// TwinCAT 3 PLC project Plc
// libraries:
//   VisuElem3DPath, 3.5.6.0 (System)
//   VisuElemMeter, 3.5.6.0 (System)
//   VisuElems, 3.5.6.10 (System)
//   VisuElemsDateTime, 3.5.6.0 (System)
//   VisuElemsSpecialControls, 3.5.6.0 (System)
//   VisuElemsWinControls, 3.5.6.0 (System)
//   VisuElemTextEditor, 3.5.6.0 (System)
//   visuinputs, 3.5.6.0 (system)
//   VisuNativeControl, 3.5.6.0 (System)
//   Tc2_DMX, * (Beckhoff Automation GmbH)
//   Tc2_IoFunctions, * (Beckhoff Automation GmbH)
//   Tc2_Standard, * (Beckhoff Automation GmbH)
//   Tc2_SUPS, * (Beckhoff Automation GmbH)
//   Tc2_System, * (Beckhoff Automation GmbH)
//   Tc2_SystemCX, * (Beckhoff Automation GmbH)
//   Tc3_Interfaces, * (Beckhoff Automation GmbH)
//   Tc3_Module, * (Beckhoff Automation GmbH)
//   VisuDialogs, * (System)
//   Tc2_Utilities,3.3.11.0,Beckhoff Automation GmbH
// project tree:
//   Data types/ E_ModeRGB.TcDUT, E_StateKompressor.TcDUT, E_RolloMode.TcDUT, E_StateAnalog.TcDUT, E_WeekDay.TcDUT, ST_AnalogScaling.TcDUT, ST_DMXRGBWCtrl.TcDUT, ST_TimeSwitchTimes.TcDUT
//   Global Variables/ Globale_Variablen.TcGVL
//   / GlobalImagePool.TcGIPO (not stored), GlobalTextList.TcGTLO, PlcTaskMain.TcTTO, Visualization Manager.TcVMO (not stored), VISU_TASK.TcTTO
//   Logger/DUTs/ ST_LogFilter.TcDUT, ST_LogMessage.TcDUT, ST_LogMessageVisu.TcDUT
//   Logger/ FB_FileWriteLogString.TcPOU, FB_Logger.TcPOU, FB_LoggerSetMsg.TcPOU, G_Logger.TcGVL
//   Logger/VISUs/ V_LoggerFilterBlack.TcVIS, V_LoggerFilterLine.TcVIS, V_LoggerFilterList.TcVIS, V_LoggerFilterWhite.TcVIS, V_LoggerModul.TcVIS, V_LoggerMsgLine.TcVIS
//   POUs/Abluftsteuerung/ FB_Abluftsteuerung.TcPOU
//   POUs/Abluftsteuerung/SubSysteme/ FB_SubAbluftMaschine.TcPOU, FB_SubAbluftTaster.TcPOU
//   POUs/EG/ FB_EGHalle.TcPOU, FB_EGBuero.TcPOU
//   POUs/KG_Raueme/ FB_WCRaum.TcPOU
//   POUs/Kompressor/ FB_KompressorSteuerung.TcPOU
//   POUs/Monitoring/ FB_LiquidMonitoring.TcPOU
//   POUs/Monitoring/Submodule/ FB_LiquidSensor.TcPOU, FB_Transor.TcPOU
//   POUs/ PLC_PRG.TcPOU
//   POUs/Temperaturen/ PRG_Temperaturen.TcPOU
//   POUs/_Grundfunktionen/ FB_Heizregler.TcPOU, FB_Heizregler_FBHR.TcPOU, FB_Kuehlregler_Kompr.TcPOU, FB_Licht.TcPOU, FB_LichtBewegungsmelder.TcPOU, FB_Rollo.TcPOU, FB_RolloGruppe.TcPOU, FB_Taster.TcPOU, FB_TasterProg.TcPOU, FB_TemperatureInput.TcPOU, FB_AnalogOutput.TcPOU, FB_TimeSwitch.TcPOU, F_diColorOfTemperature.TcPOU, F_RolDownTime.TcPOU, F_Scaling.TcPOU, F_SunRise.TcPOU
//   POUs/_Grundfunktionen/System/ FB_BK1250Diag.TcPOU, FB_SystemCX.TcPOU
//   Visualizations/Frames/ V_Dialog_Mob.TcVIS, V_Main_Mob.TcVIS, V_Main_PC.TcVIS
//   Visualizations/Module/ V_ECReset.TcVIS, V_LiquidSensorCfg.TcVIS, V_LiquidSensorState.TcVIS, V_LiquidTransorState.TcVIS, V_NumInputReal.TcVIS, V_RadioButton.TcVIS, V_TCReset.TcVIS, V_WCRaum.TcVIS, V_WeekDay.TcVIS, V_dwBitToggle.TcVIS, V_Heizung.TcVIS, V_Licht.TcVIS, V_Rol.TcVIS, V_RolGrp.TcVIS
//   Visualizations/ VisuStart.TcVIS, V_Monitoring.TcVIS, V_Logger.TcVIS, V_KomprWRG.TcVIS, V_Einstellungen.TcVIS
// real-time tasks:
//   TASK Main: cycle T#5ms, priority 21, ADS port 350
//   TASK VISU_TASK: cycle T#100000us, priority 30, ADS port 351
// I/O:
//   DEVICE Device 3 (COM Port) (disabled)
//   DEVICE Device 2 (NOV-DP-RAM) (disabled)
//   DEVICE Device 5 (CX-BK) (disabled)
//     Box 5 (CX-BK)
//   DEVICE Device 8 (RT-Ethernet Protocol) (disabled), AmsNetId 0.0.0.0.9.1
//   DEVICE CX5120 (CX-BK)
//     CXBK (CX-BK)
//   DEVICE Device 1 (EtherCAT)
// variable links:
//   Plc Instance <-> CX5120 (CX-BK)/CXBK (CX-BK)
//     PlcTaskMain Inputs/.gfbTemp11_Puffer4000_Brauchw.IiDataIn <-> AI01 Temp (KL3204)/Channel 1/Data In
//     PlcTaskMain Inputs/.gfbTemp11_Puffer4000_Brauchw.IusiState <-> AI01 Temp (KL3204)/Channel 1/State
//     PlcTaskMain Inputs/.gfbTemp12_Puffer4000_oben.IiDataIn <-> AI01 Temp (KL3204)/Channel 2/Data In
//     PlcTaskMain Inputs/.gfbTemp12_Puffer4000_oben.IusiState <-> AI01 Temp (KL3204)/Channel 2/State
//     PlcTaskMain Inputs/.gfbTemp13_Puffer4000_mitte.IiDataIn <-> AI01 Temp (KL3204)/Channel 3/Data In
//     PlcTaskMain Inputs/.gfbTemp13_Puffer4000_mitte.IusiState <-> AI01 Temp (KL3204)/Channel 3/State
//     PlcTaskMain Inputs/.gfbTemp14_Puffer4000_unten.IiDataIn <-> AI01 Temp (KL3204)/Channel 4/Data In
//     PlcTaskMain Inputs/.gfbTemp14_Puffer4000_unten.IusiState <-> AI01 Temp (KL3204)/Channel 4/State
//     PlcTaskMain Inputs/.gfbTemp21_PufferWohnh_oben.IiDataIn <-> AI02 Temp (KL3204)/Channel 1/Data In
//     PlcTaskMain Inputs/.gfbTemp21_PufferWohnh_oben.IusiState <-> AI02 Temp (KL3204)/Channel 1/State
//     PlcTaskMain Inputs/.gfbTemp22_PufferWohnh_unten.IiDataIn <-> AI02 Temp (KL3204)/Channel 2/Data In
//     PlcTaskMain Inputs/.gfbTemp22_PufferWohnh_unten.IusiState <-> AI02 Temp (KL3204)/Channel 2/State
//     PlcTaskMain Inputs/.gfbTemp23_PufferWerkst_oben.IiDataIn <-> AI02 Temp (KL3204)/Channel 3/Data In
//     PlcTaskMain Inputs/.gfbTemp23_PufferWerkst_oben.IusiState <-> AI02 Temp (KL3204)/Channel 3/State
//     PlcTaskMain Inputs/.gfbTemp24_PufferWerkst_unten.IiDataIn <-> AI02 Temp (KL3204)/Channel 4/Data In
//     PlcTaskMain Inputs/.gfbTemp24_PufferWerkst_unten.IusiState <-> AI02 Temp (KL3204)/Channel 4/State
//     PlcTaskMain Inputs/.gfbTemp31_KomprWRG_Ruecklauf.IiDataIn <-> AI03 Temp (KL3204)/Channel 1/Data In
//     PlcTaskMain Inputs/.gfbTemp31_KomprWRG_Ruecklauf.IusiState <-> AI03 Temp (KL3204)/Channel 1/State
//     PlcTaskMain Inputs/.gfbTemp32_KomprWRG_Vorlauf.IiDataIn <-> AI03 Temp (KL3204)/Channel 2/Data In
//     PlcTaskMain Inputs/.gfbTemp32_KomprWRG_Vorlauf.IusiState <-> AI03 Temp (KL3204)/Channel 2/State
//     PlcTaskMain Inputs/.gfbTemp33_WCDamen_Raum.IiDataIn <-> AI03 Temp (KL3204)/Channel 3/Data In
//     PlcTaskMain Inputs/.gfbTemp33_WCDamen_Raum.IusiState <-> AI03 Temp (KL3204)/Channel 3/State
//     PlcTaskMain Inputs/.gfbTemp34_WCHerren_Raum.IiDataIn <-> AI03 Temp (KL3204)/Channel 4/Data In
//     PlcTaskMain Inputs/.gfbTemp34_WCHerren_Raum.IusiState <-> AI03 Temp (KL3204)/Channel 4/State
//     PlcTaskMain Inputs/.gfbTemp41_Schluckbrunnen.IiDataIn <-> AI04 Temp (KL3204)/Channel 1/Data In
//     PlcTaskMain Inputs/.gfbTemp41_Schluckbrunnen.IusiState <-> AI04 Temp (KL3204)/Channel 1/State
//     PlcTaskMain Inputs/.gfbTemp42_Res.IiDataIn <-> AI04 Temp (KL3204)/Channel 2/Data In
//     PlcTaskMain Inputs/.gfbTemp43_Res.IiDataIn <-> AI04 Temp (KL3204)/Channel 3/Data In
//     PlcTaskMain Inputs/.gfbTemp44_Res.IiDataIn <-> AI04 Temp (KL3204)/Channel 4/Data In
//     PlcTaskMain Inputs/.gfbTemp42_Res.IusiState <-> AI04 Temp (KL3204)/Channel 2/State
//     PlcTaskMain Inputs/.gfbTemp43_Res.IusiState <-> AI04 Temp (KL3204)/Channel 3/State
//     PlcTaskMain Inputs/.gfbTemp44_Res.IusiState <-> AI04 Temp (KL3204)/Channel 4/State
//     PlcTaskMain Inputs/PLC_PRG.fbAbluftsteuerung1.fbAblMasch01.IbMaschineEin <-> DI04 (KL1408)/Channel 1/Input
//     PlcTaskMain Inputs/PLC_PRG.fbAbluftsteuerung2.fbAblMasch01.IbMaschineEin <-> DI04 (KL1408)/Channel 2/Input
//     PlcTaskMain Inputs/PLC_PRG.fbAbluftsteuerung1.fbAblTaster1.IbStart <-> DI04 (KL1408)/Channel 3/Input
//     PlcTaskMain Inputs/PLC_PRG.fbAbluftsteuerung2.fbAblTaster1.IbStart <-> DI04 (KL1408)/Channel 4/Input
//     PlcTaskMain Inputs/PLC_PRG.fbEGBuero.fbLichtBueroAssist.IbInBewegunsm <-> DI02 (KL1408)/Channel 6/Input
//     PlcTaskMain Inputs/PLC_PRG.fbEGBuero.fbLichtBueroChef.IbInBewegunsm <-> DI02 (KL1408)/Channel 5/Input
//     PlcTaskMain Inputs/PLC_PRG.fbEGBuero.fbLichtPausenraum.IbInBewegunsm <-> DI02 (KL1408)/Channel 4/Input
//     PlcTaskMain Inputs/PLC_PRG.fbEGHalle.IbRolloWindmesser <-> DI03 (KL1408)/Channel 5/Input
//     PlcTaskMain Inputs/PLC_PRG.fbEGHalle.fbLichtHalleAltbau.IbInBewegunsm <-> DI02 (KL1408)/Channel 2/Input
//     PlcTaskMain Inputs/PLC_PRG.fbEGHalle.fbLichtHalleAnbau.IbInBewegunsm <-> DI02 (KL1408)/Channel 3/Input
//     PlcTaskMain Inputs/PLC_PRG.fbEGHalle.fbLichtHalleNeubau.IbInBewegunsm <-> DI02 (KL1408)/Channel 1/Input
//     PlcTaskMain Inputs/PLC_PRG.fbKompressorSteuerung.IbStart <-> DI01 (KL1408)/Channel 5/Input
//     PlcTaskMain Inputs/PLC_PRG.fbKompressorSteuerung.IbStoerung <-> DI01 (KL1408)/Channel 7/Input
//     PlcTaskMain Inputs/PLC_PRG.fbKompressorSteuerung.IbStop <-> DI01 (KL1408)/Channel 6/Input
//     PlcTaskMain Inputs/PLC_PRG.fbKompressorSteuerung.fbAnalogOutUmwaelzpumpeWRG.IiDataIn <-> AO01 (KL4004)/Channel 1/Data In
//     PlcTaskMain Inputs/PLC_PRG.fbKompressorSteuerung.fbAnalogOutUmwaelzpumpeWRG.IusiState <-> AO01 (KL4004)/Channel 1/State
//     PlcTaskMain Inputs/PLC_PRG.fbWCDamen.IbLichtBewegungsmelder <-> DI03 (KL1408)/Channel 2/Input
//     PlcTaskMain Inputs/PLC_PRG.fbWCDamen.IbTasterHeizenStart <-> DI03 (KL1408)/Channel 1/Input
//     PlcTaskMain Inputs/PLC_PRG.fbWCHerren.IbLichtBewegungsmelder <-> DI03 (KL1408)/Channel 4/Input
//     PlcTaskMain Inputs/PLC_PRG.fbWCHerren.IbTasterHeizenStart <-> DI03 (KL1408)/Channel 3/Input
//     PlcTaskMain Outputs/.gfbTemp11_Puffer4000_Brauchw.QiDataOut <-> AI01 Temp (KL3204)/Channel 1/Data Out
//     PlcTaskMain Outputs/.gfbTemp11_Puffer4000_Brauchw.QusiCtrl <-> AI01 Temp (KL3204)/Channel 1/Ctrl
//     PlcTaskMain Outputs/.gfbTemp12_Puffer4000_oben.QiDataOut <-> AI01 Temp (KL3204)/Channel 2/Data Out
//     PlcTaskMain Outputs/.gfbTemp12_Puffer4000_oben.QusiCtrl <-> AI01 Temp (KL3204)/Channel 2/Ctrl
//     PlcTaskMain Outputs/.gfbTemp13_Puffer4000_mitte.QiDataOut <-> AI01 Temp (KL3204)/Channel 3/Data Out
//     PlcTaskMain Outputs/.gfbTemp13_Puffer4000_mitte.QusiCtrl <-> AI01 Temp (KL3204)/Channel 3/Ctrl
//     PlcTaskMain Outputs/.gfbTemp14_Puffer4000_unten.QiDataOut <-> AI01 Temp (KL3204)/Channel 4/Data Out
//     PlcTaskMain Outputs/.gfbTemp14_Puffer4000_unten.QusiCtrl <-> AI01 Temp (KL3204)/Channel 4/Ctrl
//     PlcTaskMain Outputs/.gfbTemp21_PufferWohnh_oben.QiDataOut <-> AI02 Temp (KL3204)/Channel 1/Data Out
//     PlcTaskMain Outputs/.gfbTemp21_PufferWohnh_oben.QusiCtrl <-> AI02 Temp (KL3204)/Channel 1/Ctrl
//     PlcTaskMain Outputs/.gfbTemp22_PufferWohnh_unten.QiDataOut <-> AI02 Temp (KL3204)/Channel 2/Data Out
//     PlcTaskMain Outputs/.gfbTemp22_PufferWohnh_unten.QusiCtrl <-> AI02 Temp (KL3204)/Channel 2/Ctrl
//     PlcTaskMain Outputs/.gfbTemp23_PufferWerkst_oben.QiDataOut <-> AI02 Temp (KL3204)/Channel 3/Data Out
//     PlcTaskMain Outputs/.gfbTemp23_PufferWerkst_oben.QusiCtrl <-> AI02 Temp (KL3204)/Channel 3/Ctrl
//     PlcTaskMain Outputs/.gfbTemp24_PufferWerkst_unten.QiDataOut <-> AI02 Temp (KL3204)/Channel 4/Data Out
//     PlcTaskMain Outputs/.gfbTemp24_PufferWerkst_unten.QusiCtrl <-> AI02 Temp (KL3204)/Channel 4/Ctrl
//     PlcTaskMain Outputs/.gfbTemp31_KomprWRG_Ruecklauf.QiDataOut <-> AI03 Temp (KL3204)/Channel 1/Data Out
//     PlcTaskMain Outputs/.gfbTemp31_KomprWRG_Ruecklauf.QusiCtrl <-> AI03 Temp (KL3204)/Channel 1/Ctrl
//     PlcTaskMain Outputs/.gfbTemp32_KomprWRG_Vorlauf.QiDataOut <-> AI03 Temp (KL3204)/Channel 2/Data Out
//     PlcTaskMain Outputs/.gfbTemp32_KomprWRG_Vorlauf.QusiCtrl <-> AI03 Temp (KL3204)/Channel 2/Ctrl
//     PlcTaskMain Outputs/.gfbTemp33_WCDamen_Raum.QiDataOut <-> AI03 Temp (KL3204)/Channel 3/Data Out
//     PlcTaskMain Outputs/.gfbTemp33_WCDamen_Raum.QusiCtrl <-> AI03 Temp (KL3204)/Channel 3/Ctrl
//     PlcTaskMain Outputs/.gfbTemp34_WCHerren_Raum.QiDataOut <-> AI03 Temp (KL3204)/Channel 4/Data Out
//     PlcTaskMain Outputs/.gfbTemp34_WCHerren_Raum.QusiCtrl <-> AI03 Temp (KL3204)/Channel 4/Ctrl
//     PlcTaskMain Outputs/.gfbTemp41_Schluckbrunnen.QiDataOut <-> AI04 Temp (KL3204)/Channel 1/Data Out
//     PlcTaskMain Outputs/.gfbTemp41_Schluckbrunnen.QusiCtrl <-> AI04 Temp (KL3204)/Channel 1/Ctrl
//     PlcTaskMain Outputs/.gfbTemp42_Res.QiDataOut <-> AI04 Temp (KL3204)/Channel 2/Data Out
//     PlcTaskMain Outputs/.gfbTemp43_Res.QiDataOut <-> AI04 Temp (KL3204)/Channel 3/Data Out
//     PlcTaskMain Outputs/.gfbTemp44_Res.QiDataOut <-> AI04 Temp (KL3204)/Channel 4/Data Out
//     PlcTaskMain Outputs/.gfbTemp42_Res.QusiCtrl <-> AI04 Temp (KL3204)/Channel 2/Ctrl
//     PlcTaskMain Outputs/.gfbTemp43_Res.QusiCtrl <-> AI04 Temp (KL3204)/Channel 3/Ctrl
//     PlcTaskMain Outputs/.gfbTemp44_Res.QusiCtrl <-> AI04 Temp (KL3204)/Channel 4/Ctrl
//     PlcTaskMain Outputs/PLC_PRG.fbAbluftsteuerung1.QbAbluftVentilator <-> DO02 (KL2408)/Channel 5/Output
//     PlcTaskMain Outputs/PLC_PRG.fbAbluftsteuerung2.QbAbluftVentilator <-> DO02 (KL2408)/Channel 6/Output
//     PlcTaskMain Outputs/PLC_PRG.fbEGBuero.fbLichtBueroAssist.QbOutLicht <-> DO04 (KL2408)/Channel 7/Output
//     PlcTaskMain Outputs/PLC_PRG.fbEGBuero.fbLichtBueroChef.QbOutLicht <-> DO04 (KL2408)/Channel 6/Output
//     PlcTaskMain Outputs/PLC_PRG.fbEGHalle.QbRolloZentralAb <-> DO04 (KL2408)/Channel 2/Output
//     PlcTaskMain Outputs/PLC_PRG.fbEGHalle.QbRolloZentralAuf <-> DO04 (KL2408)/Channel 1/Output
//     PlcTaskMain Outputs/PLC_PRG.fbEGHalle.fbLichtHalleAltbau.QbOutLicht <-> DO04 (KL2408)/Channel 4/Output
//     PlcTaskMain Outputs/PLC_PRG.fbEGHalle.fbLichtHalleAnbau.QbOutLicht <-> DO04 (KL2408)/Channel 5/Output
//     PlcTaskMain Outputs/PLC_PRG.fbEGHalle.fbLichtHalleNeubau.QbOutLicht <-> DO04 (KL2408)/Channel 3/Output
//     PlcTaskMain Outputs/PLC_PRG.fbKompressorSteuerung.QbKompressor <-> DO01 (KL2408)/Channel 6/Output
//     PlcTaskMain Outputs/PLC_PRG.fbKompressorSteuerung.QbLMStatus <-> DO01 (KL2408)/Channel 5/Output
//     PlcTaskMain Outputs/PLC_PRG.fbKompressorSteuerung.QbLufttrockner <-> DO01 (KL2408)/Channel 8/Output
//     PlcTaskMain Outputs/PLC_PRG.fbKompressorSteuerung.QbNotKompressor <-> DO01 (KL2408)/Channel 7/Output
//     PlcTaskMain Outputs/PLC_PRG.fbKompressorSteuerung.QbUmwaelzpumpeWRG <-> DO02 (KL2408)/Channel 1/Output
//     PlcTaskMain Outputs/PLC_PRG.fbKompressorSteuerung.QbUmwaelzpumpeWohnhaus <-> DO02 (KL2408)/Channel 3/Output
//     PlcTaskMain Outputs/PLC_PRG.fbKompressorSteuerung.QbVentilSchnellauflWRG <-> DO02 (KL2408)/Channel 2/Output
//     PlcTaskMain Outputs/PLC_PRG.fbKompressorSteuerung.QbVentilUmschWerkstatt <-> DO02 (KL2408)/Channel 4/Output
//     PlcTaskMain Outputs/PLC_PRG.fbKompressorSteuerung.fbAnalogOutUmwaelzpumpeWRG.QiDataOut <-> AO01 (KL4004)/Channel 1/Data Out
//     PlcTaskMain Outputs/PLC_PRG.fbKompressorSteuerung.fbAnalogOutUmwaelzpumpeWRG.QusiCtrl <-> AO01 (KL4004)/Channel 1/Ctrl
//     PlcTaskMain Outputs/PLC_PRG.fbWCDamen.QbAbluftventilator <-> DO03 (KL2408)/Channel 3/Output
//     PlcTaskMain Outputs/PLC_PRG.fbWCDamen.QbLMHeizungAktiv <-> DO03 (KL2408)/Channel 1/Output
//     PlcTaskMain Outputs/PLC_PRG.fbWCDamen.QbStellventilHeizkoerper <-> DO03 (KL2408)/Channel 2/Output
//     PlcTaskMain Outputs/PLC_PRG.fbWCHerren.QbAbluftventilator <-> DO03 (KL2408)/Channel 6/Output
//     PlcTaskMain Outputs/PLC_PRG.fbWCHerren.QbLMHeizungAktiv <-> DO03 (KL2408)/Channel 4/Output
//     PlcTaskMain Outputs/PLC_PRG.fbWCHerren.QbStellventilHeizkoerper <-> DO03 (KL2408)/Channel 5/Output
//   Plc Instance <-> Device 1 (EtherCAT)
//     PlcTaskMain Inputs/.gfbSystemCX.IuiDevState_ECMAster <-> Inputs/DevState
//   Plc Instance <-> Device 1 (EtherCAT)/Box 1 (BK1150)
//     PlcTaskMain Inputs/PLC_PRG.fbLiquidMonitoring.IbContactorResponse1 <-> DI12 (KL1408)/Channel 2/Input
//     PlcTaskMain Inputs/PLC_PRG.fbLiquidMonitoring.IbContactorResponse2 <-> DI12 (KL1408)/Channel 3/Input
//     PlcTaskMain Inputs/PLC_PRG.fbLiquidMonitoring.IbStartQuit <-> DI12 (KL1408)/Channel 1/Input
//     PlcTaskMain Inputs/PLC_PRG.fbLiquidMonitoring.fbLiquidSensor[10].IbLiquidSensor <-> DI13 (KL1408)/Channel 5/Input
//     PlcTaskMain Inputs/PLC_PRG.fbLiquidMonitoring.fbLiquidSensor[11].IbLiquidSensor <-> DI13 (KL1408)/Channel 6/Input
//     PlcTaskMain Inputs/PLC_PRG.fbLiquidMonitoring.fbLiquidSensor[12].IbLiquidSensor <-> DI13 (KL1408)/Channel 7/Input
//     PlcTaskMain Inputs/PLC_PRG.fbLiquidMonitoring.fbLiquidSensor[1].IbLiquidSensor <-> DI12 (KL1408)/Channel 4/Input
//     PlcTaskMain Inputs/PLC_PRG.fbLiquidMonitoring.fbLiquidSensor[2].IbLiquidSensor <-> DI12 (KL1408)/Channel 5/Input
//     PlcTaskMain Inputs/PLC_PRG.fbLiquidMonitoring.fbLiquidSensor[3].IbLiquidSensor <-> DI12 (KL1408)/Channel 6/Input
//     PlcTaskMain Inputs/PLC_PRG.fbLiquidMonitoring.fbLiquidSensor[4].IbLiquidSensor <-> DI12 (KL1408)/Channel 7/Input
//     PlcTaskMain Inputs/PLC_PRG.fbLiquidMonitoring.fbLiquidSensor[5].IbLiquidSensor <-> DI12 (KL1408)/Channel 8/Input
//     PlcTaskMain Inputs/PLC_PRG.fbLiquidMonitoring.fbLiquidSensor[6].IbLiquidSensor <-> DI13 (KL1408)/Channel 1/Input
//     PlcTaskMain Inputs/PLC_PRG.fbLiquidMonitoring.fbLiquidSensor[7].IbLiquidSensor <-> DI13 (KL1408)/Channel 2/Input
//     PlcTaskMain Inputs/PLC_PRG.fbLiquidMonitoring.fbLiquidSensor[8].IbLiquidSensor <-> DI13 (KL1408)/Channel 3/Input
//     PlcTaskMain Inputs/PLC_PRG.fbLiquidMonitoring.fbLiquidSensor[9].IbLiquidSensor <-> DI13 (KL1408)/Channel 4/Input
//     PlcTaskMain Outputs/PLC_PRG.fbLiquidMonitoring.QbLMStartQuit <-> DO12 (KL2408)/Channel 7/Output
//     PlcTaskMain Outputs/PLC_PRG.fbLiquidMonitoring.QbLMStatusOK <-> DO12 (KL2408)/Channel 6/Output
//     PlcTaskMain Outputs/PLC_PRG.fbLiquidMonitoring.QbStartTransor <-> DO12 (KL2408)/Channel 1/Output
//     PlcTaskMain Outputs/PLC_PRG.fbLiquidMonitoring.fbLiquidSensor[10].QbLMStatus <-> DO14 (KL2408)/Channel 2/Output
//     PlcTaskMain Outputs/PLC_PRG.fbLiquidMonitoring.fbLiquidSensor[11].QbLMStatus <-> DO14 (KL2408)/Channel 3/Output
//     PlcTaskMain Outputs/PLC_PRG.fbLiquidMonitoring.fbLiquidSensor[12].QbLMStatus <-> DO14 (KL2408)/Channel 4/Output
//     PlcTaskMain Outputs/PLC_PRG.fbLiquidMonitoring.fbLiquidSensor[1].QbLMStatus <-> DO13 (KL2408)/Channel 1/Output
//     PlcTaskMain Outputs/PLC_PRG.fbLiquidMonitoring.fbLiquidSensor[2].QbLMStatus <-> DO13 (KL2408)/Channel 2/Output
//     PlcTaskMain Outputs/PLC_PRG.fbLiquidMonitoring.fbLiquidSensor[3].QbLMStatus <-> DO13 (KL2408)/Channel 3/Output
//     PlcTaskMain Outputs/PLC_PRG.fbLiquidMonitoring.fbLiquidSensor[4].QbLMStatus <-> DO13 (KL2408)/Channel 4/Output
//     PlcTaskMain Outputs/PLC_PRG.fbLiquidMonitoring.fbLiquidSensor[5].QbLMStatus <-> DO13 (KL2408)/Channel 5/Output
//     PlcTaskMain Outputs/PLC_PRG.fbLiquidMonitoring.fbLiquidSensor[6].QbLMStatus <-> DO13 (KL2408)/Channel 6/Output
//     PlcTaskMain Outputs/PLC_PRG.fbLiquidMonitoring.fbLiquidSensor[7].QbLMStatus <-> DO13 (KL2408)/Channel 7/Output
//     PlcTaskMain Outputs/PLC_PRG.fbLiquidMonitoring.fbLiquidSensor[8].QbLMStatus <-> DO13 (KL2408)/Channel 8/Output
//     PlcTaskMain Outputs/PLC_PRG.fbLiquidMonitoring.fbLiquidSensor[9].QbLMStatus <-> DO14 (KL2408)/Channel 1/Output
//     PlcTaskMain Outputs/PLC_PRG.fbLiquidMonitoring.fbTransor[{1..4}].QbTransor <-> DO12 (KL2408)/Channel {2..5}/Output  (4 links)

CONFIGURATION Plc
    RESOURCE PLC ON TwinCAT3
        TASK PlcTaskMain(INTERVAL := T#5ms, PRIORITY := 21);
        TASK VISU_TASK(INTERVAL := T#100000us, PRIORITY := 30);
        PROGRAM PLC_PRG WITH PlcTaskMain : PLC_PRG;
        PROGRAM VisuElems_Visu_Prg WITH VISU_TASK : VisuElems.Visu_Prg;
    END_RESOURCE
END_CONFIGURATION

// ---- Data types/E_ModeRGB.TcDUT
TYPE E_ModeRGB :
(
	eModeRGB_Off,
	eModeRGB_MANUAL,
	eModeRGB_AUTO,
	eModeRGB_AUTOREVERS
);
END_TYPE

// ---- Data types/E_StateKompressor.TcDUT
TYPE E_StateKompressor :
(
	eStateKompr_AUS,
	eStateKompr_START,
	eStateKompr_AKTIV,
	eStateKompr_STOP,
	eStateKompr_STOERUNG
);
END_TYPE

// ---- Data types/E_RolloMode.TcDUT
TYPE E_RolloMode : (
	eRollo_Stop,
	eRollo_Manuell,
	eRollo_Auto,
	eRollo_Schatten);
END_TYPE

// ---- Data types/E_StateAnalog.TcDUT
TYPE E_StateAnalog : (
	eAnalog_Init,
	eAnalog_Start,
	eAnalog_LimitLow,
	eAnalog_LimitHigh,
	eAnalog_End
	);
END_TYPE

// ---- Data types/E_WeekDay.TcDUT
TYPE E_WeekDay :(
	Sonntag,
	Montag,
	Dienstag,
	Mittwoch,
	Donnerstag,
	Freitag,
	Samstag,

// folgende Eintraege sind nur zur Moduloberechnung
	Sonntag2,
	Montag2,
	Dienstag2,
	Mittwoch2,
	Donnerstag2,
	Freitag2,
	Samstag2
	);
END_TYPE

// ---- Data types/ST_AnalogScaling.TcDUT
TYPE ST_AnalogScaling :
STRUCT
	diXRef 	: DINT := 0;
	diYRef	: DINT := 2100;
	diFact	: DINT := 5000;

END_STRUCT
END_TYPE

// ---- Data types/ST_DMXRGBWCtrl.TcDUT
TYPE ST_DMXRGBWCtrl :
STRUCT
	bTickManual		: BOOL; (* Zyklus-Ticks fuer manuelle Verstellung *)
	bTickAuto			: BOOL; (* Zyklus-Ticks fuer automatische Programme *)
	rBrightness		: REAL := 1.0; (* zentraler Helligkeits-Override *)
	rRGBCtrl			: REAL; (* Steuerwert fuer den Farbton *)
	byRed					: BYTE; (* Steuerwert fuer den Farbton rot *)
	byGreen				: BYTE; (* Steuerwert fuer den Farbton grün *)
	byBlue				: BYTE; (* Steuerwert fuer den Farbton blau *)
	byWhite				: BYTE; (* Steuerwert fuer den Farbton weiss *)
	
END_STRUCT
END_TYPE

// ---- Data types/ST_TimeSwitchTimes.TcDUT
TYPE ST_TimeSwitchTimes :
STRUCT
	todHeizEin		: ARRAY[0..iTIMESWITCH_NUMOFTIMES] OF TIME_OF_DAY;
	todHeizAus		: ARRAY[0..iTIMESWITCH_NUMOFTIMES] OF TIME_OF_DAY;
	eDayOfWeekStart : ARRAY[0..iTIMESWITCH_NUMOFTIMES] OF E_WeekDay := [iTIMESWITCH_NUMOFTIMES(Montag)];
	eDayOfWeekEnd : ARRAY[0..iTIMESWITCH_NUMOFTIMES] OF E_WeekDay := [iTIMESWITCH_NUMOFTIMES(Sonntag)];

END_STRUCT
END_TYPE

// ---- Logger/DUTs/ST_LogFilter.TcDUT
TYPE ST_LogFilter :
(*
  ***************************************************************************
  ***************************************************************************
  Module owner:                 ST_EW_SW_SY, woerz 
  Keyword:                      keyword, <Feature-ID> 
  
  Description (summary): PLC Message logger filter

  ***************************************************************************
*)
STRUCT
  bEnabled : BOOL;
  szText : STRING(40);
END_STRUCT
END_TYPE

// ---- Logger/DUTs/ST_LogMessage.TcDUT
TYPE ST_LogMessage :
STRUCT
  iTyp : INT; // 0=hint 1=warning 2=error
  dtDateTime : DATE_AND_TIME;
  szPath : STRING(60);
  szMessage : STRING(80);
END_STRUCT
END_TYPE

// ---- Logger/DUTs/ST_LogMessageVisu.TcDUT
TYPE ST_LogMessageVisu :
STRUCT
	iLogId : INT;
	iTyp : INT;
	szLogMsg : STRING(160);
END_STRUCT
END_TYPE

// ---- Global Variables/Globale_Variablen.TcGVL
{attribute 'Tc2GvlVarNames'}
VAR_GLOBAL CONSTANT
	gciHeizGr			: INT := 9;
	gciHeizTimer 	: INT := 1;
	giPWMMax			: INT := 150;
	gdwPWMfast_75 : DWORD := 2000;
	gdwPWMfast_88 : DWORD := 8000;

	giNumOfAICh		: INT := 6;
	giNumOfAIGrp	: INT := 7;

	iTIMESWITCH_NUMOFTIMES : INT := 5;

END_VAR

VAR_GLOBAL
	gbTakt100ms		: BOOL;
  gdwBlink      : DWORD;

	gfbSystemCX		: FB_SystemCX := (INCFGDiagBK1250:= TRUE);

	grSunRiseFact : REAL;

	gbLichtZentralAus 	: BOOL := FALSE;
	gbLichtZentralEin 	: BOOL := FALSE;

	gbTimeRolloAb				: BOOL;
	gbTimeRolloAuf			: BOOL;

	gbTimeNacht					: BOOL;
	gbTimeTag						: BOOL;
	gbTag								: BOOL;
	gbNacht							: BOOL := TRUE;

	gbPWMTakt						: BOOL;
	giPWMTimer					: INT;
	gbHeizGruppe 				: ARRAY[0..gciHeizGr] OF BOOL;

	(* Temperatureingänge *)
	gfbTemp11_Puffer4000_Brauchw	: FB_TemperatureInput := ( (*  *)
		INrCalibFactor := 1.0,
		INrCalibOffset := 0.0);
	gfbTemp12_Puffer4000_oben			: FB_TemperatureInput := ( (*  *)
		INrCalibFactor := 1.0,
		INrCalibOffset := 0.0);
	gfbTemp13_Puffer4000_mitte		: FB_TemperatureInput := ( (*  *)
		INrCalibFactor := 1.0,
		INrCalibOffset := 0.0);
	gfbTemp14_Puffer4000_unten		: FB_TemperatureInput := ( (*  *)
		INrCalibFactor := 1.0,
		INrCalibOffset := 0.0);
	gfbTemp21_PufferWohnh_oben	: FB_TemperatureInput := ( (*  *)
		INrCalibFactor := 1.0,
		INrCalibOffset := 0.0);
	gfbTemp22_PufferWohnh_unten		: FB_TemperatureInput := ( (*  *)
		INrCalibFactor := 1.0,
		INrCalibOffset := 0.0);
	gfbTemp23_PufferWerkst_oben		: FB_TemperatureInput := ( (*  *)
		INrCalibFactor := 1.0,
		INrCalibOffset := 0.0);
	gfbTemp24_PufferWerkst_unten	: FB_TemperatureInput := ( (*  *)
		INrCalibFactor := 1.0,
		INrCalibOffset := 0.0);
	gfbTemp31_KomprWRG_Ruecklauf	: FB_TemperatureInput := ( (* Wassertemperatur WRG zum Puffer (heiss) *)
		INrCalibFactor := 1.0,
		INrCalibOffset := 0.0);
	gfbTemp32_KomprWRG_Vorlauf		: FB_TemperatureInput := ( (*  *)
		INrCalibFactor := 1.0,
		INrCalibOffset := 0.0);
	gfbTemp33_WCDamen_Raum				: FB_TemperatureInput := ( (*  *)
		INrCalibFactor := 1.0,
		INrCalibOffset := 0.0);
	gfbTemp34_WCHerren_Raum				: FB_TemperatureInput := ( (*  *)
		INrCalibFactor := 1.0,
		INrCalibOffset := 0.0);
	gfbTemp41_Schluckbrunnen			: FB_TemperatureInput := ( (*  *)
		INrCalibFactor := 1.0,
		INrCalibOffset := 0.0);
	gfbTemp42_Res									: FB_TemperatureInput := ( (*  *)
		INrCalibFactor := 1.0,
		INrCalibOffset := 0.0);
	gfbTemp43_Res									: FB_TemperatureInput := ( (*  *)
		INrCalibFactor := 1.0,
		INrCalibOffset := 0.0);
	gfbTemp44_Res									: FB_TemperatureInput := ( (*  *)
		INrCalibFactor := 1.0,
		INrCalibOffset := 0.0);

END_VAR

VAR_GLOBAL PERSISTENT
	VnvdiLichtTofKurz	: DINT := 5; (* Minuten *)
	VnvdiLichtTofLang	: DINT := 60; (* Minuten *)
	VnvstSwitchTimesLichtBWMtofLang : ST_TimeSwitchTimes; // Bewegungsmelder-Licht: Schaltzeiten fuer lange Ausschaltverzoegerung 

END_VAR

// ---- Logger/G_Logger.TcGVL
(*
  ***************************************************************************
  ***************************************************************************
  Module owner:                 ST_EW_SW_SY, woerz 
  Keyword:                      keyword, <Feature-ID> 
  
  Description (summary): PLC Message logger

  ***************************************************************************
*)
VAR_GLOBAL CONSTANT
  iMAXNUMOFMSGPERSISTENT : INT := 500; // maximum num of messages in persistent array
  iMINNUMOFMSGWRITETOFILE : INT := 100; // writing to file will start, if this num of messages are present
  iMINTIMEAFTERFILEWRITING : TIME := T#10M; // minimum waiting time, after writing to file
  iMAXNUMOFLOGFILES : INT := 3; // maximum num of log files
  diMAXNUMOFLOGITEMSPERFILE : DINT := 5000; // maximum num of log items per file
  
   // file path/name on target system (IPC)
  szLOGFILEPATH_TARGETSYSTEM : T_MaxString := 'C:\PlcLogger\'; ; 
  szLOGFILEPATH_NETWORK : T_MaxString := 'S:\Dokumente\PlcLogger\';
  
END_VAR
VAR_GLOBAL
  gfbLogger : FB_Logger;

END_VAR

// ---- POUs/PLC_PRG.TcPOU
PROGRAM PLC_PRG
VAR
	bInit							: BOOL := TRUE;

	tonCount : TON := (PT:= t#200ms);

	bSetClock  				: BOOL;
	bCopyToClockSet 	: BOOL := TRUE;
	bTimeCalc  				: BOOL;
	dtClockSet 				: DATE_AND_TIME := DT#2008-01-01-00:00;
	dwSysTimeSet			: DWORD;

	rtrigRolloAb	: R_TRIG;
	rtrigRolloAuf : R_TRIG;
	bVisuRolloAb 	: BOOL;
	bVisuRolloAuf : BOOL;

	tonTakt100ms	: TON := (PT:= t#100ms);
	tonTaktPWM	: TON := (PT:= t#5s);
	bTakt200ms	: BOOL;

	todRolloAb_i		: TIME_OF_DAY;

	dwdNacht_i			: DWORD;
	todNacht_i			: TIME_OF_DAY;
	todTag_i				: TIME_OF_DAY;

	bIn										: BOOL;
	fbTasterZentral1 			: FB_Taster;
	IbZentral1  	 AT %I* : BOOL;
	bInVisuZentral1				: BOOL;

	bVisuLichtZentralAus 	: BOOL;
	bVisuLichtZentralEin 	: BOOL;

	bLichtZentralAus 	: BOOL;
	bLichtZentralEin 	: BOOL;

(*
	fbTasterZentral2 		: FB_Taster;
	IbZentral2  AT %I*3.1	: BOOL;
	bInVisuZentral2			: BOOL;*)

	iHGr	: INT;
	iHTi	: INT;
	
	(* Funktionsbausteine ************************************)

	(* Kompressorsteuerung ***********************************)
	fbKompressorSteuerung		: FB_KompressorSteuerung;

	(* Abluft bzw. Absaugung *********************************)
	fbAbluftsteuerung1			: FB_Abluftsteuerung;
	fbAbluftsteuerung2			: FB_Abluftsteuerung;
	
  // Monitoring
  fbLiquidMonitoring : FB_LiquidMonitoring;

	(* EG-Raeume *)
  fbEGHalle : FB_EGHalle;
  fbEGBuero : FB_EGBuero;
  
	(* KG-Raeume *)
	fbWCDamen								: FB_WCRaum();
	fbWCHerren							: FB_WCRaum();
	
	
  fbLog : FB_LoggerSetMsg;
END_VAR

VAR PERSISTENT
	bSummerTime		: BOOL;

	todRolloAuf		: TIME_OF_DAY := TOD#7:30;
	todRolloAb		: TIME_OF_DAY := TOD#18:55;
	dwRolloAbMinFact_neg	: DWORD := 115;
	dwRolloAbMinFact_pos	: DWORD := 135;


	todHeizEin		: ARRAY[0..gciHeizGr,0..gciHeizTimer] OF TIME_OF_DAY :=[ TOD#0:00];
	todHeizAus		: ARRAY[0..gciHeizGr,0..gciHeizTimer] OF TIME_OF_DAY :=[ TOD#0:00];

END_VAR

IF bInit THEN
	A_Init();
END_IF
gfbSystemCX();


(* Systemuhr ***************************)
IF gfbSystemCX.OUTbNewDay
OR bTimeCalc
THEN
	(* Datum hat sich geaendert (neuer Tag) *)
	A_TimeCalculation();
	bTimeCalc := FALSE;
END_IF

(* Rollo-Timer *)
IF (todRolloAb <> TOD#00:00) THEN
	rtrigRolloAb(CLK:= (gfbSystemCX.OUTtodClockBase = todRolloAb_i));
  IF rtrigRolloAb.Q OR bVisuRolloAb THEN
    IF NOT gbTimeRolloAb THEN
      fbLog.M_AddMsgHint('Rollo AB zentral');
    END_IF
	  gbTimeRolloAb := TRUE;
	END_IF
ELSE
	gbTimeRolloAb := FALSE;
END_IF
IF (todRolloAuf <> TOD#00:00) THEN
	rtrigRolloAuf(CLK:= (gfbSystemCX.OUTtodClock = todRolloAuf));
  IF rtrigRolloAuf.Q OR bVisuRolloAuf THEN
    IF NOT gbTimeRolloAuf THEN
      fbLog.M_AddMsgHint('Rollo AUF zentral');
    END_IF
	  gbTimeRolloAuf := TRUE;
	END_IF
ELSE
	gbTimeRolloAuf := FALSE;
END_IF


(* Tag/Nacht-Timer *)
gbTimeNacht := FALSE;
gbTimeTag := FALSE;
IF (gfbSystemCX.OUTtodClockBase = todTag_i) THEN
	gbTimeTag := TRUE;
	gbTag := TRUE;
	gbNacht := FALSE;
ELSIF (gfbSystemCX.OUTtodClockBase = todNacht_i) THEN
	gbTimeNacht := TRUE;
	gbTag := FALSE;
	gbNacht := TRUE;
END_IF



(* Heizgruppen-Timer *)
FOR iHGr := 0 TO gciHeizGr DO
	gbHeizGruppe[iHGr] := FALSE;
	FOR iHTi := 0 TO gciHeizTimer DO
		IF (todHeizAus[iHGr,iHTi] <> TOD#00:00)
		AND (todHeizEin[iHGr,iHTi] <> TOD#00:00)
		AND (gfbSystemCX.OUTtodClock >= todHeizEin[iHGr,iHTi])
		AND (gfbSystemCX.OUTtodClock < todHeizAus[iHGr,iHTi])
		THEN
			gbHeizGruppe[iHGr] := TRUE;
		END_IF
	END_FOR
END_FOR

(* Taktgeber *)
gbTakt100ms := FALSE;
tonTakt100ms(IN:=TRUE);
IF 	tonTakt100ms.Q THEN
	tonTakt100ms(IN:=FALSE);
	gbTakt100ms := TRUE;
  gdwBlink := gdwBlink + 1;
END_IF;


gbPWMTakt := FALSE;
tonTaktPWM(IN:=TRUE);
IF 	tonTaktPWM.Q THEN
	tonTaktPWM(IN:=FALSE);
	gbPWMTakt := TRUE;
	giPWMTimer := giPWMTimer + 1;
	IF giPWMTimer >= giPWMMax THEN
		giPWMTimer := 0;
	END_IF
END_IF


(* Zentraltaster *)
bIn := IbZentral1 OR bInVisuZentral1;
fbTasterZentral1(bIn:= bIn);

IF fbTasterZentral1.bKlick THEN
  IF NOT bLichtZentralAus THEN
    fbLog.M_AddMsgHint('Licht Zentral Aus');
	  bLichtZentralAus := TRUE;
  END_IF
ELSIF fbTasterZentral1.bLang THEN
  IF NOT bLichtZentralAus THEN
    fbLog.M_AddMsgHint('Licht Zentral Aus');
    bLichtZentralAus := TRUE;
  END_IF
ELSE
	bLichtZentralAus := FALSE;
END_IF

gbLichtZentralAus :=
		 bLichtZentralAus
	OR bVisuLichtZentralAus;
gbLichtZentralEin :=
		 bLichtZentralEin
	OR bVisuLichtZentralEin;



gbLichtZentralAus :=
		 bLichtZentralAus
	OR bVisuLichtZentralAus;
gbLichtZentralEin :=
		 bLichtZentralEin
	OR bVisuLichtZentralEin;



gbLichtZentralAus :=
		 bLichtZentralAus
	OR bVisuLichtZentralAus;
gbLichtZentralEin :=
		 bLichtZentralEin
	OR bVisuLichtZentralEin;


(*************************************************************************)
PRG_Temperaturen();
A_FBCalls();



gfbLogger();

(* END of FB ******************************************)

ACTION A_TimeCalculation:
grSunRiseFact := F_SunRise(gfbSystemCX.OUTdDate);
todRolloAb_i := F_RolDownTime(
									rSunRise:= grSunRiseFact,
									todRef:= todRolloAb,
									dwMinFact_neg:= dwRolloAbMinFact_neg,
									dwMinFact_pos:= dwRolloAbMinFact_pos);

dwdNacht_i :=
		TOD_TO_DWORD(todRolloAb_i)
	- 3600000; (* ms = TOD#01:00 *)

todNacht_i := DWORD_TO_TOD(dwdNacht_i);
todTag_i :=
		DWORD_TO_TOD(
				88200000 (* ms = TOD#24:30 *)
			- dwdNacht_i);
END_ACTION

ACTION A_FBCalls:
(* hier werden alle FB-Instanzen aufgerufen *)

fbKompressorSteuerung();

(* Abluftsteuerung *)
fbAbluftsteuerung1();
fbAbluftsteuerung2();

// Monitoring
fbLiquidMonitoring();

(* EG-Raeume *)
fbEGHalle();
fbEGBuero();

(* Kellerraeume *)
fbWCDamen(
	IOfbTemperaturRaum := gfbTemp33_WCDamen_Raum);
fbWCHerren(
	IOfbTemperaturRaum := gfbTemp34_WCHerren_Raum);

(* END of ACTION *******************************)
END_ACTION

ACTION A_Init:
bInit := FALSE;
bTimeCalc := TRUE;
tonTakt100ms(IN:=FALSE);

(* Heizungstimer intialisieren *)
IF (todHeizEin[0,0] = TOD#0:00)
AND (todHeizAus[0,0] = TOD#0:00)
THEN
	todHeizEin[0,0] := TOD#4:45;
	todHeizAus[0,0] := TOD#12:00;
	todHeizEin[0,1] := TOD#14:00;
	todHeizAus[0,1] := TOD#19:00;

	todHeizEin[1,0] := TOD#4:50;
	todHeizAus[1,0] := TOD#20:30;

	todHeizEin[2,0] := TOD#8:00;
	todHeizAus[2,0] := TOD#12:00;
	todHeizEin[2,1] := TOD#13:00;
	todHeizAus[2,1] := TOD#17:00;

	todHeizEin[3,0] := TOD#7:30;
	todHeizAus[3,0] := TOD#11:00;
	todHeizEin[3,1] := TOD#12:45;
	todHeizAus[3,1] := TOD#18:00;

	todHeizEin[4,0] := TOD#10:00;
	todHeizAus[4,0] := TOD#13:00;
	todHeizEin[4,1] := TOD#14:00;
	todHeizAus[4,1] := TOD#19:00;

END_IF

(* END ***********************)
END_ACTION

END_PROGRAM

// ---- POUs/_Grundfunktionen/FB_Taster.TcPOU
FUNCTION_BLOCK FB_Taster
VAR_INPUT
	bIn 		: BOOL;
END_VAR

VAR_OUTPUT
	bOut	: BOOL;
	bKlick			: BOOL;
	bKlick2			: BOOL;
	bKlick3			: BOOL;
	bLang				: BOOL;
	iKlick			: INT;
END_VAR
VAR
	bKlick_i		: BOOL;

	iKlickCnt		: INT;

	tofPrell 		: TOF := (PT:= t#30ms);
	tofKlick 		: TOF := (PT:= t#400ms);
	tonLang 		: TON := (PT:= t#700ms);

	rtrigTast	 	: R_TRIG;
	ftrigKlick 	: F_TRIG;
	rtrigLang  	: R_TRIG;

END_VAR

tofPrell(IN:= bIn);
bOut := tofPrell.Q;
rtrigTast(CLK:= tofPrell.Q);
bKlick_i := rtrigTast.Q AND NOT tofKlick.Q;

tofKlick(IN:= rtrigTast.Q);
ftrigKlick(CLK:= tofKLick.Q);

IF rtrigTast.Q THEN
	iKlickCnt := iKlickCnt + 1;
END_IF

tonLang(IN:= bOut);
rtrigLang(CLK:= tonLang.Q);



(* Ausgabe *)
bKlick := bKlick_i;
IF ftrigKlick.Q THEN
	iKlick := iKlickCnt;
	bKlick2 := iKlick = 2;
	bKlick3 := iKlick = 3;
	iKlickCnt := 0;
ELSE
	iKlick := 0;
	bKlick2 := FALSE;
	bKlick3 := FALSE;
END_IF

bLang := rtrigLang.Q;

END_FUNCTION_BLOCK

// ---- POUs/Kompressor/FB_KompressorSteuerung.TcPOU
FUNCTION_BLOCK FB_KompressorSteuerung
VAR_INPUT
END_VAR
VAR_OUTPUT
END_VAR
VAR_IN_OUT
	
END_VAR
VAR
	bInit															: BOOL := TRUE;

	eState														: E_StateKompressor;
	
	IbStart										AT %I*	: BOOL;
	IbStop										AT %I*	: BOOL;
	IbStoerung								AT %I*	: BOOL;

	QbLMStatus								AT %Q*	: BOOL; (* Leuchtmelder Kompressorstatus *)
	QbKompressor							AT %Q*	: BOOL; (* Hauptkompressor *)
	QbNotKompressor						AT %Q*	: BOOL; (* Notkompressor *)
	QbLufttrockner						AT %Q*	: BOOL; (* Lufttrockner *)
	QbUmwaelzpumpeWRG					AT %Q*	: BOOL; (* Kompressor-Waermerueckgew. Umwaelzpumpe *)
	QbVentilSchnellauflWRG		AT %Q*	: BOOL; (* Umschaltventil zur Schnellaufladung des Puffers durch WRG *)
	QbUmwaelzpumpeWohnhaus		AT %Q*	: BOOL; (* Umwaelzpumpe vom Puffer zum Wohnhaus und Werkstatt *)
	QbVentilUmschWerkstatt		AT %Q*	: BOOL; (* Umschaltventil von Wohnhaus zur Werkstatt *)

	fbAnalogOutUmwaelzpumpeWRG				: FB_AnalogOutput;
	fbKuehlregler_Kompr								: FB_Kuehlregler_Kompr;
	
	tonKompressorStart								: TON := (PT:= T#300S); (* Kompressor-Startverzoegerung nach Lufttrockner *)
	tonLufttrocknerStop								: TON := (PT:= T#240S); (* Lufttrocker Nachlaufzeit nach Kompressorabschaltung *)
	tofUmwaelzpumpe										: TOF := (PT:= T#15M); (* Umwaelzpumpem Nachlaufzeit *)

	VbStart														: BOOL; (* Visu: Start *)
	VbStop														: BOOL; (* Visu: Stop *)
	bStop															: BOOL;
	rtrigStart												: R_TRIG;
	tonVisuReset											: TON := (PT:= T#2S);
	tonStartLang											: TON := (PT:= T#2S);
	bTempAnfordWohnhaus								: BOOL;
	bTempAnfordWerkstatt							: BOOL;
	
	bWRGPufferTemperatur_ValueOk			: BOOL;
	rWRGPufferTemperatur_Value				: REAL;
	
  fbLog : FB_LoggerSetMsg;
END_VAR
VAR PERSISTENT
	VrUmwaelzpumpeWRGSollwert					: REAL := 30; (* Sollwert in % *)
	VrKomprWRG_TempVorlaufSollwert		: REAL := 70; (* Kompressor-WRG Vorlauf Sollwert in °C *)
	VrKomprWRG_TempSchnellaufl				: REAL := 55; (* Kompressor-WRG Schnellaufladung bis Temparutur im Puffer oben in °C *)
	VrKomprWRG_TempUmschaltZurWohnh		: REAL := 55; (* Kompressor-WRG 4000l-Puffertemperatur, bei der auf Wohnaus umgeschaltet werden soll in °C *)
	VrKomprWRG_TempUmschaltZurWerkst	: REAL := 55; (* Kompressor-WRG Wohnh.-Puffertemperatur, bei der auf Werkstatt umgeschaltet werden soll  in °C *)
	VrKomprWRG_TempUmschaltHyst				: REAL := 3.0; (* Kompressor-WRG Temperartur-Umschalthysterese in °C *)
	VrKomprWRG_TempMinDifferenz				: REAL := 3.0; (* Kompressor-WRG Mindest-Temperaturdifferenz zwischen den Puffern in °C *)
	
	ViWRGTempSensorSelect							: INT := 3; (* Auswahl des Temperatursensors zur Steuerung der Pufferumwaelzpumpen zum Wohnhaus/Werkstatt 
			1: Puffer4000_unten
			2: Puffer4000_mitte
			3: Puffer4000_oben
			4: Puffer4000_Brauchw *)

END_VAR


bStop := IbStop OR VbStop;
rtrigStart(CLK := IbStart OR VbStart);
IF NOT IbStart
	AND NOT VbStart
OR bStop 
THEN
	tonStartLang(IN:= FALSE);
ELSE
	IF rtrigStart.Q THEN
		tonStartLang.IN := TRUE;
	END_IF	
	tonStartLang();
END_IF

tonVisuReset(IN:= VbStart OR VbStop);
IF tonVisuReset.Q THEN
	VbStart := FALSE;
	VbStop := FALSE;
END_IF

CASE eState OF

	eStateKompr_AUS:
		QbLMStatus := FALSE;
		QbKompressor := FALSE;
		QbNotKompressor := FALSE;
		QbLufttrockner := FALSE;
		tonKompressorStart(IN:= FALSE);
		tonLufttrocknerStop(IN:= FALSE);
		
		IF NOT bStop
		AND rtrigStart.Q
		THEN
      fbLog.M_AddMsgHint('Kompressor START Lufttrockner');
			eState := eStateKompr_START;
		END_IF
	
	eStateKompr_START:
		QbLufttrockner := TRUE;
		QbLMStatus := gdwBlink.2;
		tonKompressorStart(IN:= TRUE);
	
		IF bStop THEN
      fbLog.M_AddMsgHint('Kompressor STOP');
			eState := eStateKompr_AUS;
		ELSIF tonKompressorStart.Q THEN
			(* Kompressor-Startverzoegerung nach Lufttrockner *)
      fbLog.M_AddMsgHint('Kompressor aktivieren');
			eState := eStateKompr_AKTIV;
		ELSIF tonStartLang.Q THEN
			(* Kompressor direkt starten, wenn Start-Taster dauerhaft betätigt wird *)
      fbLog.M_AddMsgHint('Kompressor aktivieren (schnellstart)');
			eState := eStateKompr_AKTIV;
		END_IF
	
	eStateKompr_AKTIV:
		QbKompressor := TRUE;
		QbNotKompressor := TRUE;
		QbLMStatus := TRUE;
	
		IF bStop THEN
      fbLog.M_AddMsgHint('Kompressor STOP');
			eState := eStateKompr_STOP;
		END_IF
	
	eStateKompr_STOP:
		QbKompressor := FALSE;
		QbNotKompressor := FALSE;
		QbLMStatus := FALSE;
		tonLufttrocknerStop(IN:= TRUE);
	
		IF NOT bStop
		AND rtrigStart.Q
		THEN
			eState := eStateKompr_AKTIV;
		ELSIF tonLufttrocknerStop.Q THEN
			eState := eStateKompr_AUS;
		END_IF
	
	eStateKompr_STOERUNG: 
		IF bStop THEN
			eState := eStateKompr_AUS;
		END_IF

END_CASE


(* Kompressor-Kuehlung (Waermerueckgewinnung WRG) *)
A_Kuehlung();


(* FB END*)

ACTION A_Kuehlung:
tofUmwaelzpumpe(IN := QbKompressor);

IF gfbTemp32_KomprWRG_Vorlauf.OUTbValueOk THEN
	(* Regler fuer Kuehlung aktivieren *)
	fbKuehlregler_Kompr.INbEnable := tofUmwaelzpumpe.Q;
ELSE
	(* Isttemperatur ungueltig => Regelung nicht moeglich *)
	fbKuehlregler_Kompr.INbEnable := FALSE;
END_IF
fbKuehlregler_Kompr(
	INrTempSoll := VrKomprWRG_TempVorlaufSollwert,
	INrTempIst := gfbTemp32_KomprWRG_Vorlauf.OUTrValue);

IF tofUmwaelzpumpe.Q THEN
	(* Umwaelzpumpe WRG vom Kompressor *)
	QbUmwaelzpumpeWRG := TRUE;
	fbAnalogOutUmwaelzpumpeWRG.INbEnable := TRUE;
	IF fbKuehlregler_Kompr.INbEnable THEN
		fbAnalogOutUmwaelzpumpeWRG.INrValue :=
				fbKuehlregler_Kompr.OUTrResult / 100; 
	ELSE
		(* wenn Kuehlregeler inaktiv, dann die Umwaelzpumpe mit Festsollwert betreiben *)
		fbAnalogOutUmwaelzpumpeWRG.INrValue := 
				VrUmwaelzpumpeWRGSollwert / 100;
	END_IF
	
	(* Umschalt-Ventil fuer Schnellaufladung des 4000l-Puffers *)
	IF gfbTemp12_Puffer4000_oben.OUTbValueOk THEN
		IF (gfbTemp12_Puffer4000_oben.OUTrValue
				< (VrKomprWRG_TempSchnellaufl
					- VrKomprWRG_TempUmschaltHyst))
		THEN
			QbVentilSchnellauflWRG := TRUE;
		ELSIF (gfbTemp12_Puffer4000_oben.OUTrValue
				> VrKomprWRG_TempSchnellaufl)
		THEN
			QbVentilSchnellauflWRG := FALSE;
		END_IF
	ELSE (* Stoerung Temperatursensor *)
		QbVentilSchnellauflWRG := FALSE;
	END_IF

	(* Umwaelzpumpe zum Wohnhaus bzw. Werkstatt ***************************************************)
	(* Auswahl des Temperatursensors*)
	CASE ViWRGTempSensorSelect OF
	1: (* Puffer4000_unten *)
		bWRGPufferTemperatur_ValueOk := gfbTemp14_Puffer4000_unten.OUTbValueOk;
		rWRGPufferTemperatur_Value := gfbTemp14_Puffer4000_unten.OUTrValue;

	2: (* Puffer4000_mitte *)
		bWRGPufferTemperatur_ValueOk := gfbTemp13_Puffer4000_mitte.OUTbValueOk;
		rWRGPufferTemperatur_Value := gfbTemp13_Puffer4000_mitte.OUTrValue;

	3: (* Puffer4000_oben *)
		bWRGPufferTemperatur_ValueOk := gfbTemp12_Puffer4000_oben.OUTbValueOk;
		rWRGPufferTemperatur_Value := gfbTemp12_Puffer4000_oben.OUTrValue;

	4: (* Puffer4000_Brauchw *)
		bWRGPufferTemperatur_ValueOk := gfbTemp11_Puffer4000_Brauchw.OUTbValueOk;
		rWRGPufferTemperatur_Value := gfbTemp11_Puffer4000_Brauchw.OUTrValue;

	END_CASE

	IF bWRGPufferTemperatur_ValueOk THEN
		(* pruefen, ob die Temperaturdifferenz zw. Puffer und Wohnhaus ausreichend ist
			und damit das Laden des Wohnhauspuffers sinnvoll ist *)
		IF NOT gfbTemp22_PufferWohnh_unten.OUTbValueOk THEN
			bTempAnfordWohnhaus := FALSE;
		ELSIF bTempAnfordWohnhaus THEN
			IF (rWRGPufferTemperatur_Value
					< (gfbTemp22_PufferWohnh_unten.OUTrValue
						+ VrKomprWRG_TempMinDifferenz))
			THEN
				bTempAnfordWohnhaus := FALSE;

			ELSIF (rWRGPufferTemperatur_Value
					< (VrKomprWRG_TempUmschaltZurWohnh
							- VrKomprWRG_TempUmschaltHyst))
			THEN
				bTempAnfordWohnhaus := FALSE;
			END_IF			

		ELSIF (rWRGPufferTemperatur_Value
					> (gfbTemp22_PufferWohnh_unten.OUTrValue
						+ VrKomprWRG_TempMinDifferenz
						+ VrKomprWRG_TempUmschaltHyst))
		AND (rWRGPufferTemperatur_Value
					> VrKomprWRG_TempUmschaltZurWohnh)
		THEN
			bTempAnfordWohnhaus := TRUE;

		ELSE
			bTempAnfordWohnhaus := FALSE;
		END_IF

		(* pruefen, ob die Temperaturdifferenz zw. Puffer rund Werkstatt ausreichend ist
			und damit das Laden des Werkstattpuffers sinnvoll ist *)
		IF NOT gfbTemp24_PufferWerkst_unten.OUTbValueOk THEN
			bTempAnfordWerkstatt := FALSE;
		ELSIF bTempAnfordWerkstatt THEN
			IF (rWRGPufferTemperatur_Value
					< (gfbTemp24_PufferWerkst_unten.OUTrValue
						+ VrKomprWRG_TempMinDifferenz))
			THEN
				bTempAnfordWerkstatt := FALSE;

			ELSIF (rWRGPufferTemperatur_Value
					< (VrKomprWRG_TempUmschaltZurWerkst
							- VrKomprWRG_TempUmschaltHyst))
			THEN
				bTempAnfordWerkstatt := FALSE;
			END_IF

		ELSIF (rWRGPufferTemperatur_Value
					> (gfbTemp24_PufferWerkst_unten.OUTrValue
						+ VrKomprWRG_TempMinDifferenz
						+ VrKomprWRG_TempUmschaltHyst))
		AND (rWRGPufferTemperatur_Value
					> VrKomprWRG_TempUmschaltZurWerkst)
		THEN
			bTempAnfordWerkstatt := TRUE;

		ELSE
			bTempAnfordWerkstatt := FALSE;
		END_IF
						
		IF bTempAnfordWohnhaus THEN
			QbUmwaelzpumpeWohnhaus := TRUE;
			QbVentilUmschWerkstatt := TRUE;

		ELSIF bTempAnfordWerkstatt THEN
			QbUmwaelzpumpeWohnhaus := TRUE;
			QbVentilUmschWerkstatt := FALSE;
		
		ELSE
			QbUmwaelzpumpeWohnhaus := FALSE;
			QbVentilUmschWerkstatt := FALSE;
		END_IF
	
	ELSE (* Stoerung Temperatursensor *)
		QbUmwaelzpumpeWohnhaus := FALSE;
		QbVentilUmschWerkstatt := FALSE;
		bTempAnfordWohnhaus :=  FALSE;
		bTempAnfordWerkstatt := FALSE;
	END_IF
	
ELSE
	fbAnalogOutUmwaelzpumpeWRG.INbEnable := FALSE;
	QbUmwaelzpumpeWRG := FALSE;
	QbVentilSchnellauflWRG := FALSE;
	QbUmwaelzpumpeWohnhaus := FALSE;
	QbVentilUmschWerkstatt := FALSE;
END_IF
fbAnalogOutUmwaelzpumpeWRG();


(* END of Action *)
END_ACTION

END_FUNCTION_BLOCK

// ---- POUs/_Grundfunktionen/FB_AnalogOutput.TcPOU
FUNCTION_BLOCK FB_AnalogOutput
VAR CONSTANT
	iMAX_VALUE         				: INT   := 32760;
	iMIN_VALUE         				: INT   := 0; 
END_VAR
VAR_INPUT
	INrCalibFactor						: REAL := 1.0; (* Kalibrierungs-Faktor *)
	INrCalibOffset						: REAL := 0.0; (* Kalibrierungs-Offset *)
	
	INbEnable									: BOOL;
	INrMinValue								: REAL := 0.0;
	INrMaxValue								: REAL := 1.0;
	INrValue									: REAL; (* Ausgabewert -1.0 ... +1.0 *)
END_VAR
VAR_OUTPUT
END_VAR
VAR
	bInit											: BOOL := TRUE;
	
	IusiState					AT %I*	: USINT;
	IiDataIn 					AT %I*	: INT;
	QusiCtrl 					AT %Q*	: USINT;
	QiDataOut					AT %Q*	: INT;

	rValue										: REAL; (* Ausgabewert -1.0 ... +1.0 *)
	rMinValue									: REAL;
	rMaxValue									: REAL;

END_VAR

IF INbEnable THEN
	rMinValue := LIMIT(-1.0, INrMinValue, 1.0);
	rMaxValue := LIMIT(rMinValue, INrMaxValue, 1.0);
	
	rValue := 
			INrValue
		* INrCalibFactor
		+ INrCalibOffset;
	
	QiDataOut :=
		REAL_TO_INT(
			LIMIT(rMinValue, rValue, rMaxValue)
			* iMAX_VALUE
		);
ELSE
	QiDataOut := 0;
	
END_IF

(* END ****************************************)

END_FUNCTION_BLOCK

// ---- POUs/_Grundfunktionen/FB_Kuehlregler_Kompr.TcPOU
(* Heizregler fuer Fussbodenheizung ueber Schaltventil und 
	Ruecklauftemperaturueberwachung (Schwallbetrie)
*)
FUNCTION_BLOCK FB_Kuehlregler_Kompr
VAR_INPUT
	INbEnable				: BOOL;
	INrTempSoll			: REAL;
	INrTempIst 			: REAL;

	iPMin 					: INT := 25;
	iPMax 					: INT := 100;
	iPHeizIn				: INT := 0;
END_VAR
VAR_OUTPUT
	OUTrResult				: REAL;
END_VAR
VAR
	bInitDone					 : BOOL;

	tonCtrlCycle			: TON := (PT:=T#5S);
	bCtrlCycle				: BOOL;

	arTempIst 				: ARRAY[0..2] OF REAL;
	rTempIstAend 			: REAL;

	rTempSollOld 			: REAL;
	rTempSollAend 		: REAL;

	rTempDiff 				: REAL;

	rResult_P					: REAL;
	rResult_I					: REAL;
	rResult_Dist			: REAL;
	rResult_Dsoll			: REAL;
	rResult						: REAL;

END_VAR

VAR PERSISTENT
	VnvbManuell				: BOOL;
	VnvrResultManuell	: REAL;
	iMaxCycleTime			: INT := 3600; (* maximale Heizzykluszeit [s] bei Heizleistung 1% *)

	rkP								: REAL := 300; (* P-Regler, 1000 = 1.000 *)
	rkI								: REAL := 50; (* I-Regler, 1000 = 1.000 *)
	rkDist						: REAL := 5; (* D-Regler auf Istwert *)
	rkDsoll						: REAL := 5; (* D-Regler auf Sollwert => wirkt direkt auf I-Anteil *)

END_VAR

IF NOT bInitDone THEN
	A_Init();
END_IF

tonCtrlCycle(IN:= NOT bCtrlCycle);
bCtrlCycle := tonCtrlCycle.Q;

A_Ctrl();

(* END *******************************)

ACTION A_Init:
rTempSollOld := INrTempSoll;
arTempIst[2] := arTempIst[1];
arTempIst[1] := arTempIst[0];
arTempIst[0] := INrTempIst;
rResult_I := VnvrResultManuell * 1000;
bInitDone := TRUE;

(* END *******************************)
END_ACTION

ACTION A_Ctrl:
IF bCtrlCycle THEN
	rTempSollAend :=
			rTempSollOld
		- INrTempSoll;
	rTempSollOld := INrTempSoll;
	rTempIstAend :=
			arTempIst[2]
		- INrTempIst;
	arTempIst[2] := arTempIst[1];
	arTempIst[1] := arTempIst[0];
	arTempIst[0] := INrTempIst;
END_IF

IF VnvbManuell THEN
	rResult_I := VnvrResultManuell * 1000;
	OUTrResult := VnvrResultManuell;
	
ELSIF INbEnable
AND NOT (iPHeizIn > 0)
THEN
	IF bCtrlCycle THEN
		rResult_Dist :=
				rTempIstAend
			* rkDist;

		rResult_Dsoll :=
				rTempSollAend
			* rkDsoll;
	END_IF

	rTempDiff :=
			INrTempIst
		- INrTempSoll
		+ rResult_Dist;

	rResult_P :=
			rTempDiff
		* rkP;

	IF bCtrlCycle THEN
		rResult_I :=
				rTempDiff
			* rkI
			+ rResult_Dsoll
			+ rResult_I;
		IF (rResult_I
				> (100000 - rResult_P))
		THEN
			rResult_I :=
				(100000 - rResult_P);
		ELSIF (rResult_I < 0) THEN
			rResult_I := 0;
		END_IF
	END_IF

	rResult :=
			rResult_P
		+ rResult_I;
	OUTrResult := rResult / 1000;
END_IF

(* END *******************************)
END_ACTION

END_FUNCTION_BLOCK

// ---- Logger/FB_LoggerSetMsg.TcPOU
(*
  ***************************************************************************
  ***************************************************************************
  Module owner:                 ST_EW_SW_SY, woerz 
  Keyword:                      keyword, <Feature-ID> 
  
  Description (summary): FB to add messages to the FB_Logger

  ***************************************************************************
  #IMPORT G_Logger
*)
{attribute 'reflection'}
FUNCTION_BLOCK FB_LoggerSetMsg
VAR_INPUT
END_VAR
VAR_OUTPUT
  OUTszPath : STRING;

END_VAR
VAR
  bInit : BOOL := TRUE;

  {attribute 'instance-path'}
  {attribute 'no_init'}
  szPath  : STRING;
 
END_VAR

;

METHOD PUBLIC M_AddMsgHint
VAR_INPUT
	INszTxt : STRING;
END_VAR

M_AddMsg(0, INszTxt);
END_METHOD

METHOD PRIVATE M_Init
VAR_INPUT
END_VAR
VAR
  iMaxCutRight : INT := 10; // max num of char cutting out at end of string
  iLen : INT;
  iPosLeft : INT;
  iPosRight : INT;
END_VAR

// cut out project name (left side) and FB_LoggerSetMsg instance name (right side)
iPosLeft := FIND(szPath, '.') + 1;
iPosRight := LEN(szPath) - iMaxCutRight + FIND(RIGHT(szPath, iMaxCutRight), '.');
iLen := iPosRight - iPosLeft;
OUTszPath := MID(szPath, iLen, iPosLeft);

bInit := FALSE;
END_METHOD

METHOD PRIVATE M_AddMsg
VAR_INPUT
  INiTyp : INT;
END_VAR
VAR_IN_OUT
	IOszTxt : STRING;
END_VAR

IF bInit THEN
  M_Init();
END_IF

gfbLogger.M_SetMessage(INiTyp, OUTszPath, IOszTxt);
END_METHOD

METHOD PUBLIC M_AddMsgError
VAR_INPUT
	INszTxt : STRING;
END_VAR

M_AddMsg(2, INszTxt);
END_METHOD

METHOD PUBLIC M_AddMsgWarning
VAR_INPUT
	INszTxt : STRING;
END_VAR

M_AddMsg(1, INszTxt);
END_METHOD

END_FUNCTION_BLOCK

// ---- POUs/Abluftsteuerung/FB_Abluftsteuerung.TcPOU
FUNCTION_BLOCK FB_Abluftsteuerung
VAR CONSTANT
	diAbluftLaufzeit_RuettlerStart : DINT := 14400; (* Nach 4h = 14400sek Lauftzeit der Abluft,
																											wird der Ruettler gestartet *)
END_VAR
VAR_INPUT
END_VAR
VAR_OUTPUT
END_VAR
VAR
	bInit					: BOOL := TRUE;
	IbAbluft2_Aktiv						AT %I*	: BOOL;
	IbAbluft3_Aktiv						AT %I*	: BOOL;

	QbAbluftVentilator				AT %Q*	: BOOL;
	QbRuettler								AT %Q*	: BOOL;

	bVentilatorEin						: BOOL;
	bRuettlerEin							: BOOL;

	fbAblTaster1							: FB_SubAbluftTaster;

	fbAblMasch01							: FB_SubAbluftMaschine;
	fbAblMasch02							: FB_SubAbluftMaschine;
	fbAblMasch03							: FB_SubAbluftMaschine;
	fbAblMasch04							: FB_SubAbluftMaschine;



	tonSekundenTakt						: TON := (PT:= t#1s);
	bSekundenTakt							: BOOL;

	tofAbluftVentilator				: TOF := (PT:= T#60S);
	tofRuettlerSperrzeit			: TOF := (PT:= t#600s);
	tofRuettlerLaufzeit				: TOF := (PT:= t#60s);

END_VAR

VAR PERSISTENT
	diAbluftLaufzeit					: DINT; (* Laufzeit der Abluft in Sek. *)
END_VAR

bSekundenTakt := FALSE;
IF tonSekundenTakt.Q THEN
	tonSekundenTakt.IN := FALSE;
	bSekundenTakt := TRUE;
END_IF
tonSekundenTakt();
tonSekundenTakt.IN := TRUE;



fbAblTaster1(
	IObVentilatorEin:= bVentilatorEin,
	IObRuettlerEin:= bRuettlerEin);

fbAblMasch01(
	IObVentilatorEin:= bVentilatorEin);
	
fbAblMasch02(
	IObVentilatorEin:= bVentilatorEin);
	
fbAblMasch03(
	IObVentilatorEin:= bVentilatorEin);

fbAblMasch04(
	IObVentilatorEin:= bVentilatorEin);

	
(* Abluftventilator-Steuerung ***************************************)
tofAbluftVentilator(IN:= bVentilatorEin);
QbAbluftVentilator := tofAbluftVentilator.Q;
bVentilatorEin := FALSE;


(* Ruettler-Steuerung ***************************************)
tofRuettlerSperrzeit(
	IN:= (QbAbluftVentilator
				OR IbAbluft2_Aktiv
				OR IbAbluft3_Aktiv));

IF bSekundenTakt
AND tofRuettlerSperrzeit.IN
THEN
	diAbluftLaufzeit := diAbluftLaufzeit + 1;
END_IF

IF NOT tofRuettlerSperrzeit.Q
AND ((diAbluftLaufzeit
			> diAbluftLaufzeit_RuettlerStart)
		OR bRuettlerEin)
THEN
	tofRuettlerLaufzeit.IN := TRUE;
	diAbluftLaufzeit := 0;
END_IF
bRuettlerEin := FALSE;

tofRuettlerLaufzeit();
tofRuettlerLaufzeit.IN := FALSE;

QbRuettler := tofRuettlerLaufzeit.Q
  AND NOT tofRuettlerSperrzeit.Q;

(* END of FB **************************************)

END_FUNCTION_BLOCK

// ---- POUs/Abluftsteuerung/SubSysteme/FB_SubAbluftTaster.TcPOU
FUNCTION_BLOCK FB_SubAbluftTaster
VAR_INPUT
	INbSchieberAuf						: BOOL;
	INbRuettlerStart					: BOOL;
END_VAR
VAR_OUTPUT
	OUTbSchieber							: BOOL;
END_VAR
VAR_IN_OUT
	IObVentilatorEin					: BOOL;
	IObRuettlerEin						: BOOL;
END_VAR
VAR
	IbStart						AT %I*	: BOOL;
	IbStop						AT %I*	: BOOL;

	QbAbluftSchieber	AT %Q*	: BOOL;

	bAbluftSchieber						: BOOL;
	ftrigStart								: F_TRIG;

	tonStartLang							: TON := (PT:= t#2s);
	tofSchieber								: TOF := (PT:= T#10M);
	tofAutoStop								: TOF := (PT:= t#240m);

END_VAR

ftrigStart(CLK:= IbStart);

IF NOT IbStop
OR (bAbluftSchieber
		AND (ftrigStart.Q (* 2. Betaetigung des Start-Tasters schaltet wieder aus *)
				OR NOT tofAutoStop.Q))
THEN
	bAbluftSchieber := FALSE;

ELSIF ftrigStart.Q
AND NOT tonStartLang.Q THEN
	bAbluftSchieber := TRUE;
	tofAutoStop.IN := TRUE;

END_IF

(* Ruettler Start, wenn IbStart länger als 1 Sekunde gedrückt wird *)
tonStartLang(IN:= IbStart AND INbRuettlerStart);
IF tonStartLang.Q THEN
	IObRuettlerEin := TRUE;
END_IF



tofAutoStop();
tofAutoStop.IN := FALSE;

tofSchieber(IN:= bAbluftSchieber);
OUTbSchieber := tofSchieber.Q;
QbAbluftSchieber := OUTbSchieber OR INbSchieberAuf;

IF bAbluftSchieber THEN
	IObVentilatorEin := TRUE;
END_IF

END_FUNCTION_BLOCK

// ---- POUs/Abluftsteuerung/SubSysteme/FB_SubAbluftMaschine.TcPOU
FUNCTION_BLOCK FB_SubAbluftMaschine
VAR_INPUT
	INbSchieberAuf						: BOOL;
END_VAR
VAR_OUTPUT
	OUTbSchieber							: BOOL;
END_VAR
VAR_IN_OUT
	IObVentilatorEin					: BOOL;
END_VAR
VAR
	IbMaschineEin			AT %I*	: BOOL;
	QbAbluftSchieber	AT %Q*	: BOOL;

	bAbluftSchieber						: BOOL;
	rtrigStart								: R_TRIG;

	tofSchieber								: TOF := (PT:= T#10S); (* Abschaltverzoegerung, nachdem die Maschine ausgeschaltet wurde *)
	tofAutoStop								: TOF := (PT:= T#120M); (* automatische Abschaltung nach maximaler Betriebsdauer (Maschine durchgehend aktiv) *)

END_VAR

rtrigStart(CLK:= IbMaschineEin);

IF NOT IbMaschineEin
OR (bAbluftSchieber
		AND NOT tofAutoStop.Q)
THEN
	bAbluftSchieber := FALSE;

ELSIF rtrigStart.Q THEN
	bAbluftSchieber := TRUE;
	tofAutoStop.IN := TRUE;

END_IF

tofAutoStop();
tofAutoStop.IN := FALSE;

tofSchieber(IN:= bAbluftSchieber);
OUTbSchieber := tofSchieber.Q;
QbAbluftSchieber := OUTbSchieber OR INbSchieberAuf;

IF bAbluftSchieber THEN
	IObVentilatorEin := TRUE;
END_IF

END_FUNCTION_BLOCK

// ---- POUs/Monitoring/FB_LiquidMonitoring.TcPOU
FUNCTION_BLOCK FB_LiquidMonitoring
VAR CONSTANT
  iNUM_OF_LIQUIDSENSORS : SINT := 12;
  iNUM_OF_TRANSORS : SINT := 4;
  
END_VAR
VAR_INPUT
END_VAR
VAR_OUTPUT
END_VAR
VAR
  bInit : BOOL := TRUE;
  iId : SINT;
  
  fbLiquidSensor : ARRAY[1..iNUM_OF_LIQUIDSENSORS] OF FB_LiquidSensor;
  fbTransor : ARRAY[1..iNUM_OF_TRANSORS] OF FB_Transor;
	dwSensorState : DWORD;
	dwTransorCtrl : DWORD;

  VbStartQuit : BOOL;
  bStartQuit : BOOL;
  rtrigStartQuit : R_TRIG;
	bLMStartQuit  : BOOL;
  tonStartTransor : TON := (PT:= T#1S);
  
	// %I / %Q *********************************************************
	IbStartQuit           AT %I* : BOOL;
	IbKeySwitch           AT %I* : BOOL;
	IbContactorResponse1  AT %I* : BOOL;
	IbContactorResponse2  AT %I* : BOOL;
	QbLMStartQuit         AT %Q* : BOOL;
  QbLMStatusAlarm       AT %Q* : BOOL;
	QbLMStatusOK          AT %Q* : BOOL;
	QbStartTransor        AT %Q* : BOOL;
  
  fbLog : FB_LoggerSetMsg;
END_VAR

IF bInit THEN
  A_Init();
END_IF

rtrigStartQuit(CLK:= IbStartQuit OR VbStartQuit);
bStartQuit := rtrigStartQuit.Q AND NOT IbKeySwitch AND NOT IbContactorResponse1 AND NOT IbContactorResponse2;

dwTransorCtrl := 16#0000;
FOR iId := 1 TO iNUM_OF_LIQUIDSENSORS DO
  fbLiquidSensor[iId](
    INbQuit:= bStartQuit,
    IOdwState:= dwSensorState,
    IOdwTransorCtrl := dwTransorCtrl);
END_FOR

FOR iId := 1 TO iNUM_OF_TRANSORS DO
  fbTransor[iId](
    IOdwCtrl:= dwTransorCtrl);
END_FOR

IF (dwSensorState <> 0) THEN
  bLMStartQuit := FALSE;
  tonStartTransor.IN := FALSE;
ELSIF bLMStartQuit THEN
  IF bStartQuit THEN
    bLMStartQuit := FALSE;
    IF NOT tonStartTransor.IN THEN
      fbLog.M_AddMsgHint('Alarm quittiert, Transoren START');
      tonStartTransor.IN := TRUE;
    END_IF
	END_IF
ELSIF (dwTransorCtrl <> 0) THEN
  bLMStartQuit := TRUE;
ELSE
  IF bStartQuit THEN
    IF NOT tonStartTransor.IN THEN
      fbLog.M_AddMsgHint('Transoren START');
      tonStartTransor.IN := TRUE;
    END_IF
  END_IF
END_IF

tonStartTransor();
QbStartTransor := tonStartTransor.IN;
IF tonStartTransor.Q THEN
  tonStartTransor.IN := FALSE;
END_IF

QbLMStartQuit := bLMStartQuit AND gdwBlink.2;
QbLMStatusAlarm := bLMStartQuit OR (dwSensorState <> 0) OR (dwTransorCtrl <> 0);
QbLMStatusOK := NOT QbLMStatusAlarm;

// end of fb

ACTION A_Init:


FOR iId := 1 TO iNUM_OF_LIQUIDSENSORS DO
  fbLiquidSensor[iId].PiChannel := iId;
END_FOR

FOR iId := 1 TO iNUM_OF_TRANSORS DO
  fbTransor[iId].PiChannel := iId;
END_FOR


bInit := FALSE;

// end of action
END_ACTION

END_FUNCTION_BLOCK

// ---- POUs/Monitoring/Submodule/FB_LiquidSensor.TcPOU
FUNCTION_BLOCK FB_LiquidSensor
VAR_INPUT
  INbQuit : BOOL;
  
END_VAR
VAR_OUTPUT
END_VAR
VAR_IN_OUT
	IOdwState : DWORD;
	IOdwTransorCtrl : DWORD;
END_VAR
VAR
  iChan : SINT; // Kanalnummer im IOdwState
  bAlarm : BOOL;
  
	// %I / %Q ********************
	IbLiquidSensor  AT %I* : BOOL;
	QbLMStatus      AT %Q* : BOOL;

  fbLog : FB_LoggerSetMsg;
END_VAR
VAR PERSISTENT
  VnvdwCFGLiquidToTransor : DWORD := 16#FFFF; // Konfig. Zuordnung LiquidSensor zu Transor
  VnvszName : STRING(20);
  
END_VAR


IF IbLiquidSensor THEN
  IF NOT bAlarm THEN
    bAlarm := TRUE;
    IOdwState := SETBIT32(IOdwState, iChan);
    fbLog.M_AddMsgError('Sensor Alarm');
	END_IF
ELSIF INbQuit THEN
  IF bAlarm THEN
    bAlarm := FALSE;
    IOdwState := CLEARBIT32(IOdwState, iChan);
    fbLog.M_AddMsgHint('Alarm quittiert');
	END_IF
END_IF

QbLMStatus := bAlarm;

IF bAlarm THEN
  IOdwTransorCtrl := IOdwTransorCtrl OR VnvdwCFGLiquidToTransor;
END_IF

// end of functionblock

PROPERTY PUBLIC PiChannel : SINT
SET

IF (PiChannel >= 0) AND (PiChannel <= 31) THEN
  iChan := PiChannel;
ELSE
  iChan := 0;
END_IF
END_SET
END_PROPERTY

END_FUNCTION_BLOCK

// ---- POUs/Monitoring/Submodule/FB_Transor.TcPOU
FUNCTION_BLOCK FB_Transor
VAR_INPUT
  
END_VAR
VAR_OUTPUT
END_VAR
VAR_IN_OUT
	IOdwCtrl : DWORD;
END_VAR
VAR
  iChan : SINT; // Kanalnummer im IOdwState
  
	// %I / %Q ********************
	QbTransor       AT %Q* : BOOL;

END_VAR



QbTransor := GETBIT32(IOdwCtrl, iChan);

// end of functionblock

PROPERTY PUBLIC PiChannel : SINT
SET

IF (PiChannel >= 0) AND (PiChannel <= 31) THEN
  iChan := PiChannel;
ELSE
  iChan := 0;
END_IF
END_SET
END_PROPERTY

END_FUNCTION_BLOCK

// ---- POUs/EG/FB_EGHalle.TcPOU
FUNCTION_BLOCK FB_EGHalle
VAR_INPUT
END_VAR
VAR_OUTPUT
END_VAR
VAR_IN_OUT
	
END_VAR
VAR
	bInit					: BOOL := TRUE;

	(* %I / %Q ********************)
	IbRolloWindmesser AT %I* : BOOL;
	IbRolloZentralAuf AT %I* : BOOL;
	IbRolloZentralAb AT %I* : BOOL;
	QbRolloZentralAuf AT %Q* : BOOL;
	QbRolloZentralAb AT %Q* : BOOL;


  fbLichtHalleAltbau : FB_LichtBewegungsmelder;
  fbLichtHalleNeubau : FB_LichtBewegungsmelder;
  fbLichtHalleAnbau : FB_LichtBewegungsmelder;

  bGruppeAus : bool;
	tKurz : TIME;
	tLang : TIME;
  
END_VAR


tKurz := DINT_TO_TIME(VnvdiLichtTofKurz * 60000);
tLang := DINT_TO_TIME(VnvdiLichtTofLang * 60000);

fbLichtHalleAltbau(
	tKurz:= tKurz, 
	tLang:= tLang, 
  bGruppeAus:= bGruppeAus,
	IOstTimeSwitchTimes:= VnvstSwitchTimesLichtBWMtofLang);
  
fbLichtHalleNeubau(
	tKurz:= tKurz, 
	tLang:= tLang, 
  bGruppeAus:= bGruppeAus,
	IOstTimeSwitchTimes:= VnvstSwitchTimesLichtBWMtofLang);
  
fbLichtHalleAnbau(
	tKurz:= tKurz, 
	tLang:= tLang, 
  bGruppeAus:= bGruppeAus,
	IOstTimeSwitchTimes:= VnvstSwitchTimesLichtBWMtofLang);
  
 
(* FB END*)

END_FUNCTION_BLOCK

// ---- POUs/_Grundfunktionen/FB_LichtBewegungsmelder.TcPOU
FUNCTION_BLOCK FB_LichtBewegungsmelder
VAR_INPUT
	bEinKurz				: BOOL;
	bEinLang				: BOOL;
	bAus 						: BOOL;
	tKurz						: TIME := t#5m;
	tLang 					: TIME := t#60m;
END_VAR
VAR_OUTPUT
END_VAR
VAR_IN_OUT
	bGruppeAus : BOOL;
 	IOstTimeSwitchTimes : ST_TimeSwitchTimes;
END_VAR
VAR
	bInit 			: BOOL := TRUE;
	bInVisu			: BOOL;
	bIn					: BOOL;

	bKlickEnable	: BOOL;
	bLangEnable		: BOOL;

	(* %I / %Q ********************)
	IbInTaster		AT %I* : BOOL;
	IbInBewegunsm AT %I* : BOOL;
	QbOutLicht		AT %Q* : BOOL;

	tofEin			: TOF;

	fbTaster 		: FB_Taster;
  fbTimeSwitch : FB_TimeSwitch;
  
END_VAR

IF bInit THEN
	bKlickEnable := (tkurz <> t#0s);
	bLangEnable := (tLang <> t#0s);
	bInit := FALSE;
END_IF

fbTimeSwitch(IOstTimeSwitchTimes := IOstTimeSwitchTimes);

bIn := IbInTaster OR bInVisu;
fbTaster(bIn:= bIn);

IF IbInBewegunsm THEN
  IF fbTimeSwitch.OUTbOn THEN
    IF bKlickEnable THEN
      tofEin(IN:= TRUE, PT:= tLang);
  	END_IF
  ELSE
    IF bKlickEnable THEN
      tofEin(IN:= TRUE, PT:= tkurz);
  	END_IF
	END_IF

ELSIF bKlickEnable
AND (fbTaster.bKlick
		OR bEinKurz
		OR gbLichtZentralEin)
THEN
	tofEin(IN:= TRUE, PT:= tkurz);
ELSIF bLangEnable
AND (fbTaster.bLang
		OR bEinLang)
THEN
	tofEin(IN:= TRUE, PT:= tLang);
END_IF
tofEin(IN:= FALSE);

IF fbTaster.bLang
AND bKlickEnable
AND bLangEnable
OR bEinKurz
OR bEinLang
OR gbLichtZentralEin
OR IbInBewegunsm
THEN
	QbOutLicht := TRUE;
END_IF

IF (fbTaster.bKlick
		AND bKlickEnable)
OR (fbTaster.bLang
		AND NOT bKlickEnable
		AND bLangEnable)
THEN
	QbOutLicht := NOT QbOutLicht;
END_IF

IF QbOutLicht AND NOT tofEin.Q
OR gbLichtZentralAus OR bAus THEN
	QbOutLicht := FALSE;
END_IF

IF fbTaster.bKlick2 THEN
	bGruppeAus := TRUE;
END_IF

END_FUNCTION_BLOCK

// ---- POUs/_Grundfunktionen/FB_TimeSwitch.TcPOU
FUNCTION_BLOCK FB_TimeSwitch
VAR_INPUT
END_VAR
VAR_OUTPUT
	OUTbOn				: BOOL;
	OUTbOn_RTrig	: BOOL;
	OUTbOn_FTrig	: BOOL;
	
END_VAR
VAR_IN_OUT
	IOstTimeSwitchTimes : ST_TimeSwitchTimes;
END_VAR
VAR
	iCh						: INT;
	bOn						: BOOL;
	eDayOfWeekEnd : E_WeekDay;
	
END_VAR

bOn := FALSE;
FOR iCh := 0 TO iTIMESWITCH_NUMOFTIMES DO
	IF (IOstTimeSwitchTimes.todHeizAus[iCh] <> TOD#00:00)
	AND (IOstTimeSwitchTimes.todHeizEin[iCh] <> TOD#00:00)
	THEN
		IF (gfbSystemCX.OUTtodClock 
				>= IOstTimeSwitchTimes.todHeizEin[iCh])
		AND (gfbSystemCX.OUTtodClock 
					< IOstTimeSwitchTimes.todHeizAus[iCh])
		THEN
      IF (IOstTimeSwitchTimes.eDayOfWeekEnd[iCh] < IOstTimeSwitchTimes.eDayOfWeekStart[iCh]) THEN
        // Modulokorrektur
        eDayOfWeekEnd := IOstTimeSwitchTimes.eDayOfWeekEnd[iCh] + 7;
      ELSE
        eDayOfWeekEnd := IOstTimeSwitchTimes.eDayOfWeekEnd[iCh];
      END_IF
      IF (gfbSystemCX.OUTeDayOfWeek >= IOstTimeSwitchTimes.eDayOfWeekStart[iCh]) 
      AND (gfbSystemCX.OUTeDayOfWeek <= eDayOfWeekEnd) 
      THEN 
        bOn := TRUE;
      END_IF
		END_IF
	END_IF
END_FOR

OUTbOn_RTrig := FALSE;
OUTbOn_FTrig := FALSE;
IF NOT bOn
AND OUTbOn
THEN
	OUTbOn_FTrig := TRUE;
ELSIF bOn
AND NOT OUTbOn
THEN
	OUTbOn_RTrig := TRUE;
END_IF
OUTbOn := bOn;

(* FB END *)

END_FUNCTION_BLOCK

// ---- POUs/EG/FB_EGBuero.TcPOU
FUNCTION_BLOCK FB_EGBuero
VAR_INPUT
END_VAR
VAR_OUTPUT
END_VAR
VAR_IN_OUT
	
END_VAR
VAR
	bInit					: BOOL := TRUE;

  fbLichtBueroChef : FB_LichtBewegungsmelder;
  fbLichtBueroAssist : FB_LichtBewegungsmelder;
  fbLichtPausenraum : FB_LichtBewegungsmelder;

  bGruppeAus : bool;
	tKurz : TIME;
	tLang : TIME;
  
END_VAR


tKurz := DINT_TO_TIME(VnvdiLichtTofKurz * 60000);
tLang := DINT_TO_TIME(VnvdiLichtTofLang * 60000);
  
fbLichtBueroChef(
	tKurz:= tKurz, 
	tLang:= tLang, 
  bGruppeAus:= bGruppeAus,
	IOstTimeSwitchTimes:= VnvstSwitchTimesLichtBWMtofLang);
  
fbLichtBueroAssist(
	tKurz:= tKurz, 
	tLang:= tLang, 
  bGruppeAus:= bGruppeAus,
	IOstTimeSwitchTimes:= VnvstSwitchTimesLichtBWMtofLang);
  
fbLichtPausenraum(
	tKurz:= tKurz, 
	tLang:= tLang, 
  bGruppeAus:= bGruppeAus,
	IOstTimeSwitchTimes:= VnvstSwitchTimesLichtBWMtofLang);
  
  
(* FB END*)

END_FUNCTION_BLOCK

// ---- POUs/KG_Raueme/FB_WCRaum.TcPOU
FUNCTION_BLOCK FB_WCRaum
VAR_INPUT
END_VAR
VAR_OUTPUT
END_VAR
VAR_IN_OUT
	(* Analgoe Eingaenge ***************************)
	IOfbTemperaturRaum					: FB_TemperatureInput; (* Raumtermperatur *)
	
END_VAR
VAR
	bInit					: BOOL := TRUE;

	IbLichtBewegungsmelder		AT %I*	: BOOL;
	IbTasterHeizenStart				AT %I*	: BOOL;

	QbLMHeizungAktiv					AT %Q*	: BOOL;
	QbStellventilHeizkoerper	AT %Q*	: BOOL;
	QbAbluftventilator				AT %Q*	: BOOL;

	tofAbluftVentilator				: TOF := (PT:= T#60S);
END_VAR

VAR PERSISTENT
	VdiAbluftNachlaufzeit							: DINT := 60; (* Sekunden *)
	
END_VAR

;

(* Abluftventilator-Steuerung ***************************************)
tofAbluftVentilator(
	IN:= IbLichtBewegungsmelder,
	PT:= DINT_TO_TIME(VdiAbluftNachlaufzeit * 1000));
QbAbluftVentilator := tofAbluftVentilator.Q;


(* FB END*)

END_FUNCTION_BLOCK

// ---- POUs/_Grundfunktionen/FB_TemperatureInput.TcPOU
FUNCTION_BLOCK FB_TemperatureInput
VAR CONSTANT
	iMAX_VALUE         				: INT   := 32767; (* Drahtbruch *)
	iMIN_VALUE         				: INT   := 0; 
END_VAR
VAR_INPUT
	INrCalibFactor								: REAL := 1.0; (* Kalibrierungs-Faktor *)
	INrCalibOffset								: REAL := 0.0; (* Kalibrierungs-Offset *)
END_VAR
VAR_OUTPUT
	OUTbRangeMin 			   			: BOOL;
	OUTbRangeMax	  		   		: BOOL;
	OUTbValueOk								: BOOL;
	OUTrValue									: REAL;
END_VAR
VAR
	bInit											: BOOL := TRUE;
	
	IusiState					AT %I*	: USINT;
	IiDataIn 					AT %I*	: INT;
	QusiCtrl 					AT %Q*	: USINT;
	QiDataOut					AT %Q*	: INT;

	tonValueOk								: TON := (PT:= T#100MS);

	VdiColourOfTemperature		: DINT;
	
END_VAR

OUTbRangeMax := 
	IusiState.1
	OR (IiDataIn > iMAX_VALUE);
OUTbRangeMin := 
	IusiState.0
	OR (IiDataIn < iMIN_VALUE);

tonValueOk(
	IN:= NOT OUTbRangeMin
			AND NOT OUTbRangeMax); 	
OUTbValueOk := 
	tonValueOk.Q;

IF OUTbValueOk THEN
	OUTrValue :=
		INT_TO_REAL(IiDataIn) / 10
		* INrCalibFactor
		+ INrCalibOffset;
END_IF

VdiColourOfTemperature :=
	F_diColorOfTemperature(
		INrTempActual:= OUTrValue, 
		INrTempMin:= 20, 
		INrTempMax:= 75);
	
(* END ****************************************)

END_FUNCTION_BLOCK

// ---- POUs/_Grundfunktionen/F_diColorOfTemperature.TcPOU
FUNCTION F_diColorOfTemperature : DINT
VAR_INPUT
	INrTempActual				: REAL;
	INrTempMin					: REAL;
	INrTempMax					: REAL;
END_VAR
VAR
	rColorFactor				: REAL;
	diColor							: DINT;
	diGreen							: DINT;
	diBlue							: DINT;

END_VAR

rColorFactor := 
	16#200 / (INrTempMax - INrTempMin);

diColor :=
	REAL_TO_DINT(
		(INrTempMax 
		- INrTempActual) 
		* rColorFactor);

diGreen := LIMIT(0, diColor * 16#100, 16#FF00);
diBlue := LIMIT(0, diColor - 16#FF, 16#FF);

F_diColorOfTemperature := 16#FF0000 + diGreen + diBlue;

END_FUNCTION

// ---- POUs/Temperaturen/PRG_Temperaturen.TcPOU
PROGRAM PRG_Temperaturen
VAR
END_VAR

gfbTemp11_Puffer4000_Brauchw();
gfbTemp12_Puffer4000_oben();
gfbTemp13_Puffer4000_mitte();
gfbTemp14_Puffer4000_unten();
gfbTemp21_PufferWohnh_oben();
gfbTemp22_PufferWohnh_unten();
gfbTemp23_PufferWerkst_oben();
gfbTemp24_PufferWerkst_unten();
gfbTemp31_KomprWRG_Ruecklauf();
gfbTemp32_KomprWRG_Vorlauf();
gfbTemp33_WCDamen_Raum();
gfbTemp34_WCHerren_Raum();
gfbTemp41_Schluckbrunnen();
gfbTemp42_Res();
gfbTemp43_Res();
gfbTemp44_Res();
	
	
(* END of PRG *)

END_PROGRAM

// ---- POUs/_Grundfunktionen/F_SunRise.TcPOU
FUNCTION F_SunRise : REAL
VAR_INPUT
	dDate 				: DATE;
END_VAR
VAR CONSTANT
 (* Offset, um wieviel Tage vor Jahreswechsel der früheste Sonnenuntergang stattfindet *)
	idayOffset : INT := 25;
END_VAR
VAR
	dwDate 		: DWORD;
	dwTodRef 	: DWORD;
	rYearDay 	: REAL;

	rPi				: REAL;
	rAlpha		: REAL;

END_VAR

rPi := LREAL_TO_REAL(ACOS(-1));

dwDate := DATE_TO_DWORD(dDate);

rYearDay := DINT_TO_REAL((DWORD_TO_DINT(dwDate) MOD 31557600) / 86400 + idayOffset);

IF (rYearDay > 365) THEN
	rYearDay := rYearDay - 365;
END_IF

(* der früheste Sonnenuntergang findet etwa mitte Dez. statt, der späteste ca. Anfang Juli.
 Deshalb werden hier die ersten 210 Tage auf 180° skaliert und die restl. 155 Tage auf die 
 zweiten 180°. *)
IF (rYearDay < 210) THEN
	rAlpha := rYearDay * rPi / 210;
ELSE
	rAlpha := (rYearDay - 210) * rPi / 155 + rPi;
END_IF

(* hier wird von rAlpha nochmals rPi subtrahiert, um den Cosinus um 180° zu verschieben *)
F_SunRise := COS(rAlpha - rPi);

END_FUNCTION

// ---- POUs/_Grundfunktionen/F_RolDownTime.TcPOU
FUNCTION F_RolDownTime : TOD
VAR_INPUT
	rSunRise			: REAL;
	todRef				: TOD; (* mittlere Referenzzeit *)
	dwMinFact_neg	: DWORD;
	dwMinFact_pos	: DWORD;
END_VAR
VAR
	dwDate 		: DWORD;
	dwTodRef 	: DWORD;
	rTodRef 	: REAL;
	dwYearDay : DWORD;

	rPi				: REAL;
	rResult		: REAL;
	dwResult	: DWORD;

END_VAR

IF (rSunRise > 0) THEN
	rResult := rSunRise * DWORD_TO_REAL(dwMinFact_pos) * 60000;
ELSE
	rResult := rSunRise * DWORD_TO_REAL(dwMinFact_neg) * 60000;
END_IF

rTodRef := TOD_TO_REAL(todRef);
dwResult := REAL_TO_DWORD(rTodRef + rResult) / 1000 * 1000;

F_RolDownTime := DWORD_TO_TOD(dwResult);

END_FUNCTION

// ---- POUs/_Grundfunktionen/System/FB_SystemCX.TcPOU
FUNCTION_BLOCK FB_SystemCX
VAR_INPUT
	INCFGDiagBK1250		: BOOL;
	INstSysTimeDate	: TIMESTRUCT;
	
END_VAR
VAR_OUTPUT
	OUTbNewTime				: BOOL;
	OUTbNewMinute     : BOOL;
	OUTbNewDay				: BOOL;
	OUTbSummerTime		: BOOL;
	OUTstSysTimeDate	: TIMESTRUCT;
	OUTdtDateClock		: DATE_AND_TIME;
	OUTdDate					: DATE;
	OUTtodClockBase		: TIME_OF_DAY;
	OUTtodClock				: TIME_OF_DAY;
	OUTszClock				: STRING;
	OUTszDate					: STRING;
	OUTeDayOfWeek			: E_WeekDay;
	
END_VAR
VAR
	bInit							: BOOL := TRUE;
	bSummerTime				: BOOL;
	tonStartUp				: ton := (PT:= T#180S);

	fbUPS							: FB_S_UPS_CX51x0;
	fbBK1250Diag			: FB_BK1250Diag;

	tcRestart					: TC_Restart;
	iofDeviceReset		: IOF_DeviceReset;
	tonTcRestart			: ton := (PT:= T#3S);
	tonSetTime : ton := (PT:= T#180S);
	
	IuiDeviceId_ECMAster AT %I* : UINT; (* Device-ID EtherCAT Master *)
	IuiDevState_ECMAster AT %I* : UINT; (* EtherCAT Master *)
	QuiDevCtrl_ECMAster AT %Q* : UINT; (* EtherCAT Master *)

	(*local Windows NT time, via ADS*)
	fbNtGetTime				: NT_GetTime;
	fbNtSetTime				: NT_SetLocalTime;
	tonGetTime				: ton := (PT:=T#300MS);
	wSecond						: WORD;
	wMinute						: WORD;
	wDay							: WORD;
	bTimeCorrectStart : BOOL;
  
	VbDeviceReset			: BOOL; // EC-Master-Reset manuell (Visu)
	VbTCReset					: BOOL; // TwinCAT-Reset manuell (Visu)
	VbSetTimeStart : BOOL;
  VbSetTimeReturn : BOOL;
  VbSetTimeError : BOOL;
  
  fbLog : FB_LoggerSetMsg;
END_VAR
VAR PERSISTENT
	nvbSummerTime			: BOOL;
  nviTimeCorrectionSum : INT; // Summe Zeitkorrektur je Tag [msec]
  VnviTimeCorrectionEachDay : INT; // Zeitkorrektur je Tag [msec]
  
	nviTcRestartCnt		: INT;
	
END_VAR

IF bInit THEN
	M_Init();
END_IF

IF NOT tonStartUp.Q THEN
	tonStartUp(IN:= TRUE);
ELSE
	A_TcRestart();
END_IF

(* Ansteuerung der Sekunden-USV, damit bei Spannungsausfall die persistenten Daten gesichert werden *)
fbUPS();

(* Uhrzeit auslesen *)
fbNtGetTime();
IF NOT fbNtGetTime.BUSY THEN
	IF fbNtGetTime.START THEN
		OUTstSysTimeDate := fbNtGetTime.TIMESTR;
		fbNtGetTime.START := FALSE;
	END_IF
	tonGetTime(IN:= TRUE);
	IF tonGetTime.Q THEN
		fbNtGetTime.START := TRUE;
	END_IF
ELSE
	tonGetTime(IN:= FALSE);
END_IF

IF (OUTstSysTimeDate.wSecond
		<> wSecond)
THEN
	wSecond := OUTstSysTimeDate.wSecond;
	OUTbNewTime := TRUE;
	OUTdtDateClock := SYSTEMTIME_TO_DT(TIMESTR:= OUTstSysTimeDate);
	OUTtodClockBase := DT_TO_TOD(OUTdtDateClock);
	IF OUTbSummerTime THEN
		(* waehrend der Sommerzeit eine Stunde addieren +3600s *)
		OUTtodClock := DWORD_TO_TOD(TOD_TO_DWORD(OUTtodClockBase) + 3600000);
	ELSE
		OUTtodClock := OUTtodClockBase;
	END_IF
		
	OUTszClock := MID(TOD_TO_STRING(OUTtodClock), 8, 5);
	M_Summertime();
ELSE
	OUTbNewTime := FALSE;
END_IF

IF (OUTstSysTimeDate.wMinute <> wMinute) THEN
  wMinute := OUTstSysTimeDate.wMinute;
  OUTbNewMinute := TRUE;
ELSE
  OUTbNewMinute := FALSE;  
END_IF


IF (OUTstSysTimeDate.wDay
		<> wDay)
THEN
	wDay := OUTstSysTimeDate.wDay;
	OUTbNewDay := TRUE;
	OUTeDayOfWeek := WORD_TO_INT(OUTstSysTimeDate.wDayOfWeek);
	OUTdDate := DT_TO_DATE(OUTdtDateClock);
	OUTszDate := MID(DATE_TO_STRING(OUTdDate), 10, 3);
ELSE
	OUTbNewDay := FALSE;
END_IF


// Datum Uhrzeit einstellen
IF tonSetTime.Q THEN
  VbSetTimeStart := FALSE;
ELSIF VbSetTimeStart THEN
  IF NOT tonSetTime.IN THEN
    fbNtSetTime(START := FALSE);
    INstSysTimeDate := OUTstSysTimeDate;
    INstSysTimeDate.wSecond := 0;
    INstSysTimeDate.wMilliseconds := 0;
	END_IF
  IF VbSetTimeReturn THEN
    fbNtSetTime(START := TRUE, TIMESTR := INstSysTimeDate);
    IF NOT fbNtSetTime.BUSY THEN
      IF NOT fbNtSetTime.ERR THEN
        VbSetTimeStart := FALSE;
      ELSE
        VbSetTimeError := TRUE;
        VbSetTimeReturn := FALSE;
      END_IF
      fbNtSetTime(START := FALSE);
    END_IF
	END_IF
ELSE
  VbSetTimeReturn := FALSE;
  VbSetTimeError := FALSE;
END_IF
tonSetTime(IN:= VbSetTimeStart);

// automatische Uhrzeitkorrektur
IF (VnviTimeCorrectionEachDay <> 0) THEN
  IF OUTbNewDay THEN
    nviTimeCorrectionSum := nviTimeCorrectionSum
      + VnviTimeCorrectionEachDay;
    fbNtSetTime(START := FALSE);
	END_IF
  IF OUTbNewMinute THEN
    // Korrektur wird i.d.R. um 00:01Uhr durchgefuehrt
    IF ABS(nviTimeCorrectionSum >= 10000) THEN
      // Korrektur hat 10s erreicht
      INstSysTimeDate := OUTstSysTimeDate;
        IF (nviTimeCorrectionSum >= 10000) THEN
          // Korrektur + 10s
          INstSysTimeDate.wSecond := INstSysTimeDate.wSecond + 10;
          IF (INstSysTimeDate.wSecond > 59) THEN
            INstSysTimeDate.wSecond := 0;
            INstSysTimeDate.wMinute := INstSysTimeDate.wMinute + 1;
            IF (INstSysTimeDate.wMinute > 59) THEN
              INstSysTimeDate.wMinute := 0;
              INstSysTimeDate.wHour := INstSysTimeDate.wHour + 1;
              IF (INstSysTimeDate.wHour > 23) THEN
                INstSysTimeDate.wHour := 0;
              END_IF
            END_IF
          END_IF
        ELSE
          // Korrektur - 10s
          IF (INstSysTimeDate.wSecond >= 10) THEN
            INstSysTimeDate.wSecond := INstSysTimeDate.wSecond - 10;
          ELSIF (INstSysTimeDate.wMinute > 0) THEN
            INstSysTimeDate.wSecond := INstSysTimeDate.wSecond + 60 - 10;
            INstSysTimeDate.wMinute := INstSysTimeDate.wMinute - 1;
          END_IF
				END_IF
        IF (INstSysTimeDate.wMinute >= 0) AND (INstSysTimeDate.wMinute < 60) THEN
          // Korrektur nur bei gueltigem Zeitwert durchfuehren
          bTimeCorrectStart := TRUE;
        END_IF
    END_IF
	END_IF

  IF bTimeCorrectStart THEN
    fbNtSetTime(START := TRUE, TIMESTR := INstSysTimeDate);
    IF NOT fbNtSetTime.BUSY THEN
      bTimeCorrectStart := FALSE;
      IF NOT fbNtSetTime.ERR THEN
        IF (nviTimeCorrectionSum >= 10000) THEN
          nviTimeCorrectionSum := nviTimeCorrectionSum - 10000;
        ELSE
          nviTimeCorrectionSum := nviTimeCorrectionSum + 10000;
  			END_IF
			END_IF
      fbNtSetTime(START := FALSE);
  	END_IF
	END_IF
ELSE
  bTimeCorrectStart := FALSE;
  nviTimeCorrectionSum := 0;
END_IF


(* END *****************************************)

ACTION A_TcRestart:

IF INCFGDiagBK1250 THEN
	fbBK1250Diag();
END_IF

IF tcRestart.RESTART THEN
	// TwinCAT-Restart durchführen
	tcRestart();
	IF NOT tcRestart.BUSY OR tcRestart.ERR THEN
		tcRestart(RESTART:= FALSE);
		tonTcRestart.IN := TRUE;
	END_IF
	
ELSIF iofDeviceReset.RESET THEN
	// EtherCAT-Master RESET durchführen
	iofDeviceReset();
	IF NOT iofDeviceReset.BUSY OR iofDeviceReset.ERR THEN
		iofDeviceReset(RESET:= FALSE);
		tonTcRestart.IN := TRUE;
	END_IF
	
ELSIF NOT tonTcRestart.IN THEN
	IF fbBK1250Diag.OUTbError THEN
    nviTcRestartCnt := nviTcRestartCnt + 1;
    fbLog.M_AddMsgError(CONCAT('EC-Master-Reset autom., BK1250-State= ', UINT_TO_STRING(fbBK1250Diag.OUTuiCouplterState)));
		iofDeviceReset(RESET:= TRUE);
	ELSIF VbDeviceReset THEN
    fbLog.M_AddMsgWarning(CONCAT('EC-Master-Reset manuell, BK1250-State= ', UINT_TO_STRING(fbBK1250Diag.OUTuiCouplterState)));
		iofDeviceReset(RESET:= TRUE);

	ELSIF VbTCReset THEN
    fbLog.M_AddMsgWarning(CONCAT('EC-Master-Reset manuell, BK1250-State= ', UINT_TO_STRING(fbBK1250Diag.OUTuiCouplterState)));
		tcRestart(RESTART:= TRUE);
		
	END_IF
	
END_IF

tonTcRestart();
IF tonTcRestart.Q THEN
	VbTCReset := FALSE;
	VbDeviceReset := FALSE;
	tonTcRestart.IN := FALSE;
END_IF
END_ACTION

ACTION M_Init:
bInit := FALSE;

tcRestart(
	NETID:= '', 
	RESTART:= FALSE, 
	TMOUT:= );

iofDeviceReset(
	NETID:= '',
	DEVICEID:= IuiDeviceId_ECMAster, 
	RESET:= FALSE,  
	TMOUT:= );
	
(* Ansteuerung der Sekunden-USV, damit bei Spannungsausfall die persistenten Daten gesichert werden *)
fbUPS(
	sNetID:= '', 
	iPLCPort:= 851, 
	iUPSPort:= 16#588, 
	tTimeout:= DEFAULT_ADS_TIMEOUT, 
	eUpsMode:= eSUPS_WrPersistData_Shutdown, 
	ePersistentMode:= SPDM_2PASS, 
	tRecoverTime:= T#10S);

fbNtGetTime.NETID := ''; (*local*)
fbNtSetTime.NETID := ''; (*local*)

tonStartUp(IN:= FALSE);

OUTbSummerTime := nvbSummerTime;
	
(* END *****************************************)
END_ACTION

ACTION M_Summertime:

IF (WORD_TO_INT(OUTstSysTimeDate.wDayOfWeek) = Sonntag) THEN
	IF nvbSummerTime THEN
		IF (OUTtodClockBase = TOD#2:00) THEN
			IF (OUTstSysTimeDate.wMonth = 10)
			AND (OUTstSysTimeDate.wDay >= 25)
			THEN
				nvbSummerTime := FALSE;
			END_IF
		END_IF
	ELSE
		IF (OUTtodClockBase = TOD#2:00) THEN
			IF (OUTstSysTimeDate.wMonth = 3)
			AND (OUTstSysTimeDate.wDay >= 25)
			THEN
				nvbSummerTime := TRUE;
			END_IF
		END_IF
	END_IF
END_IF
OUTbSummerTime := nvbSummerTime;

(* END *****************************************)
END_ACTION

END_FUNCTION_BLOCK

// ---- POUs/_Grundfunktionen/System/FB_BK1250Diag.TcPOU
FUNCTION_BLOCK FB_BK1250Diag
VAR_INPUT
END_VAR
VAR_OUTPUT
	OUTbStateOK : BOOL;
	OUTbError : BOOL;
	OUTuiCouplterState : UINT;
	
END_VAR
VAR
	IuiCouplterState AT %I* : UINT;
	IbWcState AT %I* : BOOL;
	
	tonError : ton := (PT:=T#100ms);
	
END_VAR

OUTuiCouplterState := IuiCouplterState;

IF OUTuiCouplterState > 0 THEN
	tonError.IN := TRUE;
ELSIF IbWcState THEN
	tonError.IN := TRUE;
ELSE
	tonError.IN := FALSE;
END_IF

OUTbStateOK := NOT tonError.IN;
tonError();
OUTbError := tonError.Q;

END_FUNCTION_BLOCK

// ---- Logger/FB_Logger.TcPOU
FUNCTION_BLOCK FB_Logger
VAR CONSTANT
  iMAXNUMOFMSGVISU : INT := 11; // maximum num of messges in PLC-Visu list 
  iMAXNUMOFFILTER : INT := 3; // maximum num of terms in filter text
  iMAXNUMOFFILTERSTORE : INT := 10;

  aszMSGTYP : ARRAY[0..2] OF STRING(5) := ['Hint', 'Warn', 'Error'];
  
END_VAR
VAR_INPUT
  INbFileWritingEnable : BOOL := TRUE;
  INbWriteToFileAndClose : BOOL;
  INbCloseFile : BOOL;
  
END_VAR
VAR_OUTPUT
  OUTbFileOpen : BOOL;
  
END_VAR
VAR
  bInit : BOOL := TRUE;
  bSetInitMessage : BOOL;
  iPathLenMax : INT := 30;
  iProgVersion : INT;

  fbLog : FB_LoggerSetMsg;
  
  // Write to File
  bInitFileWriter : BOOL := TRUE;
  bInitPathNetwork : BOOL := FALSE;
  iStateFileWriter : INT;
  fbFileWriteLogString : FB_FileWriteLogString;
  szFileName : STRING;
  tonWaitFileWriting : TON;
  iFileWriterNumOfMsgsOpen : INT;
  iFileWriterErrorState : INT;
	iLogIdFileWriter : INT;
  bWriteToFileStart : BOOL;
  bCloseFileAndWait : BOOL;
  bWriteToFileStartVisible : BOOL; // Button bVisuWriteToFileStart anzeigen
  bVisuInitPathNetwork : BOOL;
 	bVisuWriteToFileStart : BOOL := FALSE;

  
  // PLC-Visu
  iVisuState : INT;
  bVisuStart : BOOL;
  bVisuAutoStart : BOOL;
  bVisuPrevPage : BOOL;
  bVisuPrevPageInVisible : BOOL;
  bVisuNextPage : BOOL;
  bVisuNextPageInVisible : BOOL;
  bVisuDone : BOOL;
  bVisuError : BOOL;
  iVisuLogId : INT;
  iVisuLogIdStart : INT;
  iVisuLogIdIsLastMsg : INT; // LogId im Visu-Array entspricht der letzten Meldung
  iVisuGetMsgId : INT;
  iVisuCnt : INT;
  tonVisu : TON := (PT:=T#3M);
  bVisuFilterResult : BOOL;
  bVisuNothingFound : BOOL;
  iVisuFilterListVisible : INT;
  bVisuFilterWhiteEnable : BOOL;
  bVisuFilterBlackEnable : BOOL;
  bVisuFilterWhiteMode_OR : BOOL := TRUE; // combine filterterms with AND/OR (0/1)
	szVisuFilterWhite : STRING(80);
	szVisuFilterBlack : STRING(80);
  astVisuFilterWhite : ARRAY[1..iMAXNUMOFFILTER] OF ST_LogFilter;
  astVisuFilterBlack : ARRAY[1..iMAXNUMOFFILTER] OF ST_LogFilter;
  iVisuFilterMsgTypInput : INT;
  iVisuFilterMsgTyp : INT;

  szVisuString : STRING(120);
  astVisuLogMsg : ARRAY[1..iMAXNUMOFMSGVISU] OF ST_LogMessageVisu;
  
END_VAR
VAR PERSISTENT
	nviLogId : INT;
	nviLogIdFileWriter : INT;
	anvstLogMsg : ARRAY[0..G_Logger.iMAXNUMOFMSGPERSISTENT] OF ST_LogMessage;

	anvszVisuFilter : ARRAY[0..iMAXNUMOFFILTERSTORE] OF STRING(80);
  nvstVisuActualMessage : ST_LogMessageVisu;
  
  nvbVisuFileWritingEnable : BOOL := TRUE;

END_VAR

IF bInit THEN
  M_Init();
END_IF
IF bSetInitMessage THEN
  M_SetInitMessage();
END_IF


// file writer *********************************************
A_FileWriting();


// visualisation list **************************************
tonVisu();
CASE iVisuState OF
0: // off
  bVisuDone := FALSE;
  bVisuPrevPageInVisible := TRUE;
  bVisuNextPageInVisible := TRUE;
  iVisuFilterListVisible := 0;
  IF bVisuStart THEN
    tonVisu(IN:= FALSE);
    iVisuState := iVisuState + 1;
	END_IF
  
1: // init page
  tonVisu.IN := TRUE;
  iVisuLogId := 0;
  iVisuCnt := -1; // search direction backward
  iVisuLogIdIsLastMsg := 0;
  bVisuDone := FALSE;
  bVisuPrevPage := FALSE;
  bVisuNextPage := FALSE;
  bVisuPrevPageInVisible := TRUE;
  bVisuNextPageInVisible := TRUE;
  iVisuFilterListVisible := 0;
  bVisuError := FALSE;
  bVisuAutoStart := TRUE;
  iVisuLogIdStart := nviLogId;
  iVisuGetMsgId := nviLogId;
  iVisuFilterMsgTyp := iVisuFilterMsgTypInput;  
  M_ParseFilter(szVisuFilterWhite, astVisuFilterWhite);
  M_ParseFilter(szVisuFilterBlack, astVisuFilterBlack);
  bVisuNothingFound := TRUE;
  iVisuState := iVisuState + 1;

2: // clear page
  iVisuLogId := 0;
  iVisuState := iVisuState + 1;

3: // clear page
  bVisuPrevPageInVisible := TRUE;
  bVisuNextPageInVisible := TRUE;
  iVisuLogId := iVisuLogId + 1;
  IF (iVisuLogId <= iMAXNUMOFMSGVISU) THEN
    astVisuLogMsg[iVisuLogId].iLogId := 0;
    astVisuLogMsg[iVisuLogId].iTyp := 0;
    astVisuLogMsg[iVisuLogId].szLogMsg := '';
  ELSE
    IF (iVisuCnt > 0) THEN
      iVisuLogId := iMAXNUMOFMSGVISU;
    ELSE
      iVisuLogId := 1;
		END_IF
    iVisuState := iVisuState + 1;
  END_IF

4: // create page
  IF (iVisuLogId > 0) AND (iVisuLogId <= iMAXNUMOFMSGVISU) THEN
    IF (iVisuGetMsgId < 1) AND (iVisuGetMsgId > G_Logger.iMAXNUMOFMSGPERSISTENT) THEN
      iVisuState := 90;
    ELSE
      
      IF (anvstLogMsg[iVisuGetMsgId].iTyp >= iVisuFilterMsgTyp) THEN
        // FilterMsgTyp TRUE
        
        IF M_GetMsgString(INiLogId:= iVisuGetMsgId, IOszTarget:= szVisuString) THEN
          bVisuFilterResult := TRUE;
          IF bVisuFilterWhiteEnable THEN
            IF NOT M_CheckFilter(0, szVisuString, astVisuFilterWhite) THEN
              bVisuFilterResult := FALSE;
            END_IF
          END_IF
          IF bVisuFilterBlackEnable THEN
            IF NOT M_CheckFilter(1, szVisuString, astVisuFilterBlack) THEN
              bVisuFilterResult := FALSE;
            END_IF
          END_IF
  
          IF bVisuFilterResult THEN
            // copy message to Visu list
            bVisuNothingFound := FALSE;
            astVisuLogMsg[iVisuLogId].iLogId := iVisuGetMsgId;
            astVisuLogMsg[iVisuLogId].iTyp := anvstLogMsg[iVisuGetMsgId].iTyp;
            astVisuLogMsg[iVisuLogId].szLogMsg := szVisuString;
            IF (iVisuGetMsgId = nviLogId) THEN
              iVisuLogIdIsLastMsg := iVisuLogId;
            END_IF
            iVisuLogId := iVisuLogId - iVisuCnt;
          END_IF
        END_IF
      END_IF

      // check, if search complete or next entry
      IF (iVisuCnt > 0) AND ((iVisuGetMsgId = nviLogId)) THEN
        // forward search complete
        bVisuPrevPageInVisible := FALSE;
        bVisuAutoStart := TRUE;
        iVisuState := 100;
    
      ELSE
        iVisuGetMsgId := iVisuGetMsgId + iVisuCnt;
        IF (iVisuGetMsgId < 1) THEN
          iVisuGetMsgId := G_Logger.iMAXNUMOFMSGPERSISTENT;
        ELSIF (iVisuGetMsgId > G_Logger.iMAXNUMOFMSGPERSISTENT) THEN
          iVisuGetMsgId := 1;
        END_IF
        IF (iVisuCnt < 0) AND ((iVisuGetMsgId = nviLogId)) THEN
          // backward search complete
          IF NOT bVisuAutoStart THEN
            bVisuNextPageInVisible := FALSE;
          END_IF
          iVisuState := 100;
        END_IF
      END_IF
  
		END_IF
  ELSE
    // visu list full 
    bVisuPrevPageInVisible := FALSE;
    bVisuNextPageInVisible := FALSE;
    iVisuState := 100;
	END_IF

90: // error
  bVisuError := TRUE;
  bVisuStart := FALSE;
  iVisuState := 0;


100: // done
  bVisuStart := FALSE;
  bVisuDone := TRUE;
  bVisuPrevPage := FALSE;
  bVisuNextPage := FALSE;
  IF bVisuNothingFound OR (iVisuLogIdIsLastMsg > 0) THEN
    bVisuNextPageInVisible := TRUE;
	END_IF
  iVisuState := iVisuState + 1;

101: // select command
  IF tonVisu.Q THEN
    iVisuState := 0;
	END_IF
  
  IF bVisuPrevPage AND (astVisuLogMsg[iMAXNUMOFMSGVISU].iLogId > 0) THEN
    iVisuCnt := -1; // search direction backwards
    iVisuGetMsgId := astVisuLogMsg[iMAXNUMOFMSGVISU].iLogId;
    iVisuState := 102;
  ELSIF bVisuNextPage AND (astVisuLogMsg[1].iLogId > 0) THEN
    iVisuCnt := 1; // search direction forward
    iVisuGetMsgId := astVisuLogMsg[1].iLogId;
    iVisuState := 102;
    
  ELSIF bVisuStart THEN
    // page refresh
    iVisuState := 0;

  ELSIF bVisuAutoStart THEN
    IF (iVisuLogIdStart <> nviLogId) THEN
      // new messages available => page refresh
      bVisuStart := TRUE;
      iVisuState := 1;
    ELSIF (iVisuFilterMsgTyp <> iVisuFilterMsgTypInput) THEN
      // filter message typ changed => page refresh
      bVisuStart := TRUE;
      iVisuState := 0;
  	END_IF
	END_IF
  
102: // select next/prev page
  iVisuLogIdIsLastMsg := 0;
  bVisuDone := FALSE;
  bVisuAutoStart := FALSE;
  iVisuState := 2;

END_CASE

METHOD PRIVATE M_GetMsgStringCSV : BOOL
VAR_INPUT
  INiLogId : INT;
END_VAR
VAR_IN_OUT
  IOszTarget : STRING(120);
END_VAR
VAR
  szTyp : STRING(5);
  
END_VAR

M_GetMsgStringCSV := FALSE;
IF (INiLogId > 0) AND (INiLogId <= G_Logger.iMAXNUMOFMSGPERSISTENT) THEN
  IF NOT (anvstLogMsg[INiLogId].szMessage = '') THEN
    IF (anvstLogMsg[INiLogId].iTyp >= 0) AND (anvstLogMsg[INiLogId].iTyp <= 2) THEN
      szTyp := aszMSGTYP[anvstLogMsg[INiLogId].iTyp];
    ELSE
      szTyp := INT_TO_STRING(anvstLogMsg[INiLogId].iTyp);
    END_IF
  
    IOszTarget :=
      CONCAT(szTyp,
        CONCAT(';',
          CONCAT(MID(DT_TO_STRING(anvstLogMsg[INiLogId].dtDateTime), 19, 4),
            CONCAT(';',
              CONCAT(anvstLogMsg[INiLogId].szPath,
                CONCAT(';', anvstLogMsg[INiLogId].szMessage))))));
    M_GetMsgStringCSV := TRUE;
  END_IF
END_IF
END_METHOD

ACTION A_FileWriting:

IF bInitFileWriter THEN
  fbFileWriteLogString.INiMaxLogFiles := G_Logger.iMAXNUMOFLOGFILES;
  fbFileWriteLogString.INdiMaxLogItems := G_Logger.diMAXNUMOFLOGITEMSPERFILE; 
  fbFileWriteLogString.INszNetId := ''; // HMIAgstMachineInfo.szAMS_Net_Id;
  szFileName := 'PlcLog';
  IF bInitPathNetwork THEN
    fbFileWriteLogString.INszFileName := CONCAT(G_Logger.szLOGFILEPATH_NETWORK, szFileName);
  ELSE
    fbFileWriteLogString.INszFileName := CONCAT(G_Logger.szLOGFILEPATH_TARGETSYSTEM, szFileName);
  END_IF
  bVisuInitPathNetwork := bInitPathNetwork;

  fbFileWriteLogString.INszHeadLine := 'Typ;Date and Time;PLC path;Message';
  tonWaitFileWriting(IN:= FALSE, PT:= G_Logger.iMINTIMEAFTERFILEWRITING);
  iStateFileWriter := 0;
  
  bInitFileWriter := FALSE;
END_IF


// close file by INPUT 
IF (iStateFileWriter > 0) THEN
  iFileWriterNumOfMsgsOpen := nviLogId - nviLogIdFileWriter;
  IF (iFileWriterNumOfMsgsOpen < 0) THEN
    iFileWriterNumOfMsgsOpen := iFileWriterNumOfMsgsOpen + G_Logger.iMAXNUMOFMSGPERSISTENT;
	END_IF

  IF (iStateFileWriter < 120) THEN
    IF INbCloseFile OR NOT INbFileWritingEnable OR NOT nvbVisuFileWritingEnable THEN
      iStateFileWriter := 120;
    END_IF
    bWriteToFileStart := bVisuWriteToFileStart OR INbWriteToFileAndClose;
  END_IF
END_IF

CASE iStateFileWriter OF
0: // enabled ?
  fbFileWriteLogString.INbWrite := FALSE;
  fbFileWriteLogString.INbClose := FALSE;
  bWriteToFileStartVisible := FALSE;
  bVisuWriteToFileStart := FALSE;

  IF INbFileWritingEnable AND nvbVisuFileWritingEnable THEN
    iStateFileWriter := iStateFileWriter + 1;
	END_IF

1: // init
  tonWaitFileWriting(IN:= FALSE);
  iStateFileWriter := iStateFileWriter + 1;

2: // wait min time after last write process
  bWriteToFileStartVisible := TRUE;

  bCloseFileAndWait := INbCloseFile OR INbWriteToFileAndClose
      OR (bVisuInitPathNetwork XOR bInitPathNetwork);
  
  tonWaitFileWriting(IN:= TRUE);
  IF tonWaitFileWriting.Q OR bWriteToFileStart THEN
    IF (iFileWriterNumOfMsgsOpen >= G_Logger.iMINNUMOFMSGWRITETOFILE) THEN
      bWriteToFileStartVisible := FALSE;
      iStateFileWriter := 10;
    ELSIF (iFileWriterNumOfMsgsOpen > 1) AND bWriteToFileStart THEN
      iStateFileWriter := 10;
    ELSIF bCloseFileAndWait THEN
      iStateFileWriter := 120;
    END_IF
	END_IF

10: // start writing to file
  OUTbFileOpen := TRUE;
  IF fbFileWriteLogString.OUTbError THEN
    iStateFileWriter := 90;

  ELSIF NOT fbFileWriteLogString.OUTbBusy THEN
    iLogIdFileWriter := nviLogIdFileWriter + 1;
    IF (iLogIdFileWriter > G_Logger.iMAXNUMOFMSGPERSISTENT) THEN
      iLogIdFileWriter := 1;
    END_IF
    IF M_GetMsgStringCSV(iLogIdFileWriter, fbFileWriteLogString.INszWriteLine) THEN
      fbFileWriteLogString.INbWrite := TRUE;
      iStateFileWriter := iStateFileWriter + 1;
    END_IF
	END_IF

11: // write busy
  IF NOT fbFileWriteLogString.OUTbBusy THEN
    IF fbFileWriteLogString.OUTbError THEN
      iStateFileWriter := 90;
    ELSE
      nviLogIdFileWriter := iLogIdFileWriter;
      IF (nviLogIdFileWriter <> nviLogId) THEN
        iStateFileWriter := 10; // next message
      ELSE
        // all messages written
        iStateFileWriter := 100;
      END_IF
   	END_IF
    fbFileWriteLogString.INbWrite := FALSE;
	END_IF

  
90: // error
  iFileWriterErrorState := fbFileWriteLogString.OUTiStateError;
  OUTbFileOpen := FALSE;
  IF (iFileWriterErrorState < 30) THEN
    // errror while FileOpen => repeat with local path
    bInitPathNetwork := FALSE;
    bInitFileWriter := TRUE;
	END_IF
  iStateFileWriter := 0;
  
  
100: // done
  fbFileWriteLogString.INbWrite := FALSE;
  bVisuWriteToFileStart := FALSE;
  iStateFileWriter := 120;


120: // close file ***********************************************
  fbFileWriteLogString.INbWrite := FALSE;
  fbFileWriteLogString.INbClose := TRUE;
  bWriteToFileStartVisible := FALSE;
  iStateFileWriter := iStateFileWriter + 1;

121: // wait close file
  IF NOT fbFileWriteLogString.OUTbBusy THEN    
    fbFileWriteLogString.INbClose := FALSE;
    OUTbFileOpen := FALSE;
    tonWaitFileWriting(IN:= FALSE);
    bWriteToFileStartVisible := TRUE;
    iStateFileWriter := iStateFileWriter + 1;
	END_IF

122: // wait after close to avoid file access while data backup
  IF bVisuInitPathNetwork XOR bInitPathNetwork THEN
    bInitFileWriter := FALSE;
	END_IF

  tonWaitFileWriting(IN:= NOT INbCloseFile AND NOT INbWriteToFileAndClose);
  IF tonWaitFileWriting.Q OR NOT bCloseFileAndWait THEN
    iStateFileWriter := 0;
	END_IF
  
END_CASE
 
fbFileWriteLogString();
END_ACTION

METHOD PRIVATE M_ParseFilter : BOOL
VAR_IN_OUT
  IOszFilterTerm : STRING(80);
  IOastFilter : ARRAY[1..iMAXNUMOFFILTER] OF ST_LogFilter;
END_VAR
VAR
  iFor : INT;
  iPosSep : INT;
  iLen : INT;
  szFilterTerm : STRING(80);
END_VAR

FOR iFor := 1 TO iMAXNUMOFFILTER DO
  IOastFilter[iFor].bEnabled := FALSE;
END_FOR

IF NOT (IOszFilterTerm = '') THEN
  szFilterTerm := IOszFilterTerm;  
  FOR iFor := 1 TO iMAXNUMOFFILTER DO
    iPosSep := FIND(szFilterTerm, ';');
    IF (iPosSep > 0) THEN
      iLen := iPosSep - 1;
    ELSE
      iLen := 40;
		END_IF
    IOastFilter[iFor].szText := MID(szFilterTerm, iLen, 1);
    IOastFilter[iFor].bEnabled :=  NOT (IOastFilter[iFor].szText = '');
    IF (iPosSep > 0) THEN
      szFilterTerm := MID(szFilterTerm, 40, iPosSep + 1); 
    ELSE
      EXIT;
		END_IF
  END_FOR
END_IF
END_METHOD

METHOD PRIVATE M_CheckFilter : BOOL
VAR_INPUT
  iMode : INT; // 0= white, 1= black
END_VAR
VAR_INPUT
  IOszText : STRING(80);
  IOastFilter : ARRAY[1..iMAXNUMOFFILTER] OF ST_LogFilter;
END_VAR
VAR
  iFor : INT;
  iResult : INT;
  bCheckResultOR : BOOL;
  bResultOR : BOOL;
END_VAR

M_CheckFilter := TRUE;
bResultOR := FALSE;
bCheckResultOR := FALSE;

FOR iFor := 1 TO iMAXNUMOFFILTER DO
  IF IOastFilter[iFor].bEnabled THEN
    iResult := FIND(IOszText, IOastFilter[iFor].szText);
    IF (iMode = 0) THEN
      // search mode white
      IF bVisuFilterWhiteMode_OR THEN
        // search mode OR
        bCheckResultOR := TRUE;
        IF (iResult > 0) THEN
          bResultOR := TRUE;
				END_IF
      ELSIF (iResult = 0) THEN
        // search mode AND
        M_CheckFilter := FALSE;
        EXIT;
      END_IF
    ELSIF (iMode = 1) AND (iResult > 0) THEN
      // search mode black
      M_CheckFilter := FALSE;
      EXIT;
		END_IF
	END_IF
END_FOR
 
IF bCheckResultOR AND NOT bResultOR THEN
  M_CheckFilter := FALSE;
END_IF
END_METHOD

METHOD PRIVATE M_GetMsgString : BOOL
VAR_INPUT
  INiLogId : INT;
END_VAR
VAR_IN_OUT
  IOszTarget : STRING(120);
END_VAR

M_GetMsgString := FALSE;
IF (INiLogId > 0) AND (INiLogId <= G_Logger.iMAXNUMOFMSGPERSISTENT) THEN
  IF NOT (anvstLogMsg[INiLogId].szMessage = '') THEN  
    IOszTarget :=
      CONCAT(MID(DT_TO_STRING(anvstLogMsg[INiLogId].dtDateTime), 19, 4),
        CONCAT(' ',
          CONCAT(anvstLogMsg[INiLogId].szPath,
            CONCAT(': ', anvstLogMsg[INiLogId].szMessage))));
    M_GetMsgString := TRUE;
  END_IF
END_IF
END_METHOD

METHOD PRIVATE M_SetInitMessage
VAR_INPUT
END_VAR

IF (gfbSystemCX.OUTdtDateClock > DT#1970-01-01-00:00) THEN
  fbLog.M_AddMsgWarning(
    INszTxt := 'PLC-Init after restart');
  bSetInitMessage := FALSE;
END_IF
END_METHOD

METHOD PRIVATE M_Init
VAR_INPUT
END_VAR
VAR
  iId : INT;
END_VAR

iPathLenMax := SIZEOF(anvstLogMsg[nviLogId].szPath) - 1;
bVisuInitPathNetwork := bInitPathNetwork;

bSetInitMessage := TRUE;

bInit := FALSE;
END_METHOD

METHOD PUBLIC M_SetMessage
VAR_INPUT
	INiTyp : INT;
END_VAR
VAR_IN_OUT
	IOszPath : STRING;
	IOszLogTxt : STRING;
END_VAR

nviLogId := nviLogId + 1;
IF (nviLogId > G_Logger.iMAXNUMOFMSGPERSISTENT) THEN
	nviLogId := 1;
END_IF
anvstLogMsg[nviLogId].iTyp := INiTyp;
anvstLogMsg[nviLogId].dtDateTime := gfbSystemCX.OUTdtDateClock;
anvstLogMsg[nviLogId].szPath := RIGHT(IOszPath, iPathLenMax);
anvstLogMsg[nviLogId].szMessage := IOszLogTxt;

nvstVisuActualMessage.iLogId := nviLogId;
nvstVisuActualMessage.iTyp := INiTyp;
M_GetMsgString(nviLogId, nvstVisuActualMessage.szLogMsg);

IF (nviLogId = nviLogIdFileWriter) THEN
  nviLogIdFileWriter := nviLogIdFileWriter + 1;
  IF (nviLogIdFileWriter > G_Logger.iMAXNUMOFMSGPERSISTENT) THEN
    nviLogIdFileWriter := 1;
  END_IF
END_IF
END_METHOD

END_FUNCTION_BLOCK

// ---- Logger/FB_FileWriteLogString.TcPOU
(*
  ***************************************************************************
  ***************************************************************************
  Module owner:                 Woerz 
  
  Description (summary): Function block for writing strings to logger files.

  Description (detailed):
  =======================  

  ***************************************************************************
*)

FUNCTION_BLOCK FB_FileWriteLogString
VAR CONSTANT
  tADSTIMEOUT : TIME := T#5S;	// ads timeout

END_VAR
VAR_INPUT
  // configuration inputs, no change after init
  INiMaxLogFiles : INT := 2;
  INdiMaxLogItems : DINT := 500;
  INszNetId : T_AmsNetId; // TwinCAT network address of the source file
  INszFileName : T_MaxString; // source file path and name
  INszFileNameExtension : STRING(5) := '.csv';

  // control inputs
  INbSimulation : BOOL;
	INbWrite : BOOL;
	INbClose : BOOL;
  INszHeadLine : T_MaxString;
  INszWriteLine : T_MaxString;

END_VAR

VAR_OUTPUT
  OUTbBusy : BOOL;
	OUTbError : BOOL;
	OUTbDone : BOOL;
	OUTiStateError : INT;
	OUTudiErrId : UDINT;

END_VAR

VAR
  iState : INT;
  iStateTemp : INT;
	bWriteDone : BOOL;
	bCloseDone : BOOL;
	bPutHeadline : BOOL;

  uiDestFile : UINT;
  
  tonWriteTime : TON;
  
  fbFileOpen : FB_FileOpen;
  fbFileClose : FB_FileClose;
  fbFilePuts : FB_FilePuts;

END_VAR

VAR PERSISTENT
  nvbFileNotComplete : BOOL;
  nviFileNameIndex : INT;
  nvdiLinePos : DINT;
  
END_VAR



CASE iState OF
  
0: // init
  A_Reset();
  IF (nviFileNameIndex <= 0)
  OR (nviFileNameIndex > INiMaxLogFiles) 
  THEN
    nviFileNameIndex := 0;
    nvbFileNotComplete := FALSE;
	END_IF
  OUTbBusy := FALSE;
  OUTbError := FALSE;
  OUTbDone := FALSE;
  OUTudiErrId := 0;
  uiDestFile := 0;
  iState := 1;

1: // wait for command  
  IF INbClose THEN
    IF NOT (uiDestFile = 0) THEN
      OUTiStateError := 0;
      iState := 80;
    END_IF
    
  ELSIF INbWrite THEN
    OUTbBusy := TRUE;
    OUTiStateError := 0;
    IF (uiDestFile = 0) THEN
      iState := 10; // file open
    ELSE
      iState := 20; // put string line to file
    END_IF
  END_IF


10:
  IF NOT fbFileOpen.bExecute THEN
    fbFileOpen.sNetId := INszNetId;
    IF nvbFileNotComplete THEN
      // actual file-index not complete => append to file
      fbFileOpen.nMode := FOPEN_MODEAPPEND OR FOPEN_MODEPLUS OR FOPEN_MODETEXT;
    ELSE
      // open new file or overwrite existing
      fbFileOpen.nMode := FOPEN_MODEWRITE OR FOPEN_MODEPLUS OR FOPEN_MODETEXT;
      nviFileNameIndex := nviFileNameIndex + 1;
      IF (nviFileNameIndex > INiMaxLogFiles) THEN
        nviFileNameIndex := 1;
			END_IF
      nvdiLinePos := 0;
    END_IF
    fbFileOpen.sPathName := CONCAT(INszFileName, CONCAT('_', CONCAT(INT_TO_STRING(nviFileNameIndex), INszFileNameExtension)));
    fbFileOpen.ePath := PATH_GENERIC;
    fbFileOpen.tTimeout := tAdsTimeout;
  END_IF

  fbFileOpen(bExecute := TRUE);
  IF NOT fbFileOpen.bBusy THEN
    IF fbFileOpen.bError THEN
      OUTudiErrId := fbFileOpen.nErrId;
      OUTiStateError := iState;
      nvbFileNotComplete := FALSE;
      iState := 90;
    ELSE
      uiDestFile := fbFileOpen.hFile;
      fbFilePuts.hFile := fbFileOpen.hFile;
      bPutHeadline := NOT nvbFileNotComplete AND NOT (INszHeadLine = '');
      iState := 20;
    END_IF
  END_IF


20: // put string line to file ************************************
  IF NOT fbFilePuts.bExecute THEN
    fbFilePuts.sNetId := fbFileOpen.sNetId;
    fbFilePuts.hFile := uiDestFile;
    IF bPutHeadline THEN
      fbFilePuts.sLine := CONCAT(INszHeadLine, '$N'); // new file => put headline first
    ELSE
      fbFilePuts.sLine := CONCAT(INszWriteLine, '$N');
    END_IF
    fbFilePuts.tTimeout := tAdsTimeOut;
  END_IF

  fbFilePuts(bExecute := TRUE);
  IF NOT fbFilePuts.bBusy THEN
    IF fbFilePuts.bError THEN
      OUTudiErrId := fbFilePuts.nErrId;
      OUTiStateError := iState;
      iState := 80;
    ELSE
      bWriteDone := TRUE;
      IF INbClose THEN
        iState := 80;
      ELSE
        nvbFileNotComplete := TRUE;
        nvdiLinePos := nvdiLinePos + 1;
        IF bPutHeadline THEN
          bPutHeadline := FALSE;
          fbFilePuts(bExecute := FALSE);
        ELSE
          iState := 100;
        END_IF
			END_IF
    END_IF
  END_IF

  
80: // close file ***********************************************
  IF NOT fbFileClose.bExecute THEN
    fbFileClose.sNetId := fbFileOpen.sNetId;
    fbFileClose.hFile := uiDestFile;
    fbFileClose.tTimeout := tAdsTimeOut;
  END_IF

  fbFileClose(bExecute := TRUE);
  IF NOT fbFileClose.bBusy THEN
    uiDestFile := 0;
    bCloseDone := TRUE;
    IF fbFileClose.bError THEN
      OUTudiErrId := fbFileClose.nErrId;
      OUTiStateError := iState;
      iState := 90;
    ELSE
      iState := 100;
    END_IF
  END_IF


90: // error ***********************************************
  OUTbBusy := FALSE;
  OUTbDone := FALSE;
  OUTbError := TRUE;
  IF NOT INbClose AND NOT INbWrite THEN
    OUTbError := FALSE;
    OUTiStateError := 0;
    iState := 1;
  END_IF
  
100:
  OUTbBusy := FALSE;
  OUTbDone := TRUE;

  IF (uiDestFile > 0) AND (nvdiLinePos >= INdiMaxLogItems) THEN
    // max num of logitems reached => close file
    nvbFileNotComplete := FALSE;
    iState := 80;
    
  ELSIF (uiDestFile > 0) AND INbClose AND NOT bCloseDone THEN
    iState := 80; // close file
    
	ELSIF NOT INbClose AND NOT INbWrite THEN
    OUTbDone := FALSE;
    iState := 1;
  END_IF
    
END_CASE

IF (iState > 1) AND (iState < 90) THEN
  OUTbBusy := TRUE;
  OUTbDone := FALSE;
  bCloseDone := FALSE;
END_IF

IF (iState <> iStateTemp) THEN
  iStateTemp := iState;
  A_Reset();
END_IF

ACTION A_Reset:

fbFileOpen(bExecute := FALSE);
fbFileClose(bExecute := FALSE);
fbFilePuts(bExecute := FALSE);
END_ACTION

END_FUNCTION_BLOCK

